# B&R Automation Studio project NAELD004C00R10L518F00 (part 51)

#### Act_LinkAction.st
```iecst
(** 2019-04-09 **)
ACTION Act_LinkAction:

	IF p_bLinkOpsRun = TRUE THEN
		//	p_eAct ACCESS p_OpsTravULMtrPshrAct;
		IF p_bLinkPullConvPullerExtCtrl
			AND p_bLinkPullConvPullerRetCtrl = FALSE
			AND p_bExtSen = FALSE
			THEN
				p_eAct := MtrPshrActExt;

		ELSIF p_bLinkPullConvPullerExtCtrl = FALSE
			AND p_bLinkPullConvPullerRetCtrl
			AND p_bRetSen = FALSE
			THEN
				p_eAct := MtrPshrActRet;

		ELSE
				p_eAct := MtrPshrActIdle;
		END_IF

	ELSIF p_bManual = TRUE THEN
//		IF p_UIMtrPshrAct = MtrPshrActStop THEN
//			p_eAct := MtrPshrActStop;
//		ELSE
			IF p_bLinkPullConvPullerExtCtrl
				AND p_bLinkPullConvPullerRetCtrl = FALSE
				AND p_bExtSen = FALSE
				THEN
				p_eAct := MtrPshrActExt;

			ELSIF p_bLinkPullConvPullerExtCtrl = FALSE
				AND p_bLinkPullConvPullerRetCtrl
				AND p_bRetSen = FALSE
				THEN
				p_eAct := MtrPshrActRet;

			ELSE
				p_eAct := MtrPshrActIdle;
			END_IF
//		END_IF

	ELSE
		p_eAct := MtrPshrActIdle;
	END_IF

END_ACTION
```

#### Act_Main.st
```iecst
(** 2019-06-17 **)
ACTION Act_Main:

	IF eStatOld <> eStat THEN
		bMtrSpdSlw	:= FALSE;

		fbMtrBrkOffDlyTm(IN := FALSE);
		fbMtrPshrExtChk(bEn := FALSE);
		fbMtrPshrRetChk(bEn := FALSE);

		IF eStatOld <> MtrPshrActIdle
			AND eStatOld <> MtrPshrActSetExt
			AND eStatOld <> MtrPshrActRstExt
			AND eStatOld <> MtrPshrActSetRet
			AND eStatOld <> MtrPshrActRstRet
			AND eStatOld <> MtrPshrActSetSpdBit0
			AND eStatOld <> MtrPshrActRstSpdBit0
			AND eStatOld <> MtrPshrActSetSpdBit1
			AND eStatOld <> MtrPshrActRstSpdBit1
			AND eStatOld <> MtrPshrActSetSpdBit2
			AND eStatOld <> MtrPshrActRstSpdBit2
			AND eStatOld <> MtrPshrActSetSigOn
			AND eStatOld <> MtrPshrActRstSigOn
			AND eStatOld <> MtrPshrActSetBrake
			AND eStatOld <> MtrPshrActRstBrake
			AND eStatOld <> MtrPshrActSetAlmRst
			AND eStatOld <> MtrPshrActRstAlmRst
			AND eStatOld <> MtrPshrActSetAll
			AND eStatOld <> MtrPshrActRstAll THEN

			bCW			:= FALSE;
			bCCW		:= FALSE;
			bSpdBinBit0	:= FALSE;
			bSpdBinBit1	:= FALSE;
			bSpdBinBit2	:= FALSE;
			bSigOn		:= FALSE;
			bBrake		:= FALSE;
			bAlmRst		:= FALSE;

		END_IF

		sStatTxt	:= a_sStatText[eStat];

		eStatOld	:= eStat;

		eStatus		:= Busy;
	END_IF

	//Main
	CASE eStat OF

		MtrPshrActIdle:
			IF EDGENEG(p_bManual) THEN
				bCW			:= FALSE;
				bCCW		:= FALSE;
				bSpdBinBit0	:= FALSE;
				bSpdBinBit1	:= FALSE;
				bSpdBinBit2	:= FALSE;
				bSigOn		:= FALSE;
				bBrake		:= FALSE;
				bAlmRst		:= FALSE;
			END_IF

			eStatus	:= Idle;

		MtrPshrActExt:
			IF eStatus = Idle OR eStatus = Busy THEN
				eStatus	:= Busy;

				//Motor Torque
				IF (p_bRetSen OR p_bRetSlowSen)AND NOT(bMtrSpdSlw) THEN
					iAnalogTorque	:= ((DINT_TO_INT(p_diStartTorque) * iMtrVolt) / 100);
				ELSIF bMtrSpdSlw THEN
					iAnalogTorque	:= ((DINT_TO_INT(p_diExtTorque) * iMtrVolt) / 100);
				END_IF

				IF iAnalogTorque < 1500 THEN
					iAnalogTorque	:= 1500;
				END_IF

				//Motor Speed
				IF p_bExtSlowSen = TRUE THEN
					bMtrSpdSlw	:= TRUE;
				END_IF

				IF bMtrSpdSlw = TRUE THEN
					diMtrSpd	:= p_diExtSlowSpd *usiPercent/100;
				ELSE
					diMtrSpd	:= p_diExtNomSpd *usiPercent/100;
				END_IF

				CASE diMtrSpd OF
					1:
						bSpdBinBit0	:= FALSE;
						bSpdBinBit1	:= FALSE;
						bSpdBinBit2	:= FALSE;
					2:
						bSpdBinBit0	:= TRUE;
						bSpdBinBit1	:= FALSE;
						bSpdBinBit2	:= FALSE;
					3:
						bSpdBinBit0	:= FALSE;
						bSpdBinBit1	:= TRUE;
						bSpdBinBit2	:= FALSE;
					4:
						bSpdBinBit0	:= TRUE;
						bSpdBinBit1	:= TRUE;
						bSpdBinBit2	:= FALSE;
					5:
						bSpdBinBit0	:= FALSE;
						bSpdBinBit1	:= FALSE;
						bSpdBinBit2	:= TRUE;
					6:
						bSpdBinBit0	:= TRUE;
						bSpdBinBit1	:= FALSE;
						bSpdBinBit2	:= TRUE;
					7:
						bSpdBinBit0	:= FALSE;
						bSpdBinBit1	:= TRUE;
						bSpdBinBit2	:= TRUE;
					8:
						bSpdBinBit0	:= TRUE;
						bSpdBinBit1	:= TRUE;
						bSpdBinBit2	:= TRUE;
				END_CASE

				//Motor On
				bSigOn	:= FALSE;
				bBrake	:= TRUE;

				IF p_bDir = TRUE THEN
					bCW		:= TRUE;
				ELSE
					bCCW	:= TRUE;
				END_IF

				//Checking Extend
				fbMtrPshrExtChk.bExtSen		:= p_bExtSen;
				fbMtrPshrExtChk.bRetSen		:= p_bRetSen;
				fbMtrPshrExtChk.bExtSafety	:= p_bExtSafetySen;

				fbMtrPshrExtChk(bEn := TRUE);

				IF fbMtrPshrExtChk.udiStatus = 0 THEN

					bSigOn	:= TRUE;
					bBrake	:= FALSE;
					bCW		:= FALSE;
					bCCW	:= FALSE;

					fbMtrBrkOffDlyTm(IN := TRUE);

					IF fbMtrBrkOffDlyTm.Q = TRUE THEN
						fbMtrBrkOffDlyTm(IN := FALSE);

						bCW			:= FALSE;
						bCCW		:= FALSE;
						bSpdBinBit0	:= FALSE;
						bSpdBinBit1	:= FALSE;
						bSpdBinBit2	:= FALSE;
						bSigOn		:= FALSE;
						bBrake		:= FALSE;

						bExtended	:= TRUE;
						eStatus		:= Done;
					END_IF

				ELSIF fbMtrPshrExtChk.udiStatus < 65534 THEN

					bCW			:= FALSE;
					bCCW		:= FALSE;
					bSpdBinBit0	:= FALSE;
					bSpdBinBit1	:= FALSE;
					bSpdBinBit2	:= FALSE;
					bSigOn		:= TRUE;
					bBrake		:= FALSE;

					bExtended	:= FALSE;
					eStatus		:= Error;

					IF fbMtrPshrExtChk.udiStatus = 1506 THEN
						udiStatus	:= 10000;	//Pusher Retract Sensor Off Time Out In Extend Check While Pusher Extend
					ELSIF fbMtrPshrExtChk.udiStatus = 1503 THEN
						udiStatus	:= 10001;	//Pusher Extend Sensor On Time Out In Extend Check While Pusher Extend
					ELSIF fbMtrPshrExtChk.udiStatus = 1507 THEN
						udiStatus	:= 10002;	//Pusher Extend Safety Sensor Error In Extend Check While Pusher Extend
					ELSE
						udiStatus	:= fbMtrPshrExtChk.udiStatus;
					END_IF

				END_IF

			END_IF

		MtrPshrActRet:
			IF eStatus = Idle OR eStatus = Busy THEN
				eStatus	:= Busy;

				//Motor Torque
				IF (p_bExtSen OR p_bExtSlowSen) AND NOT(bMtrSpdSlw) THEN
					iAnalogTorque	:= ((DINT_TO_INT(p_diStartTorque) * iMtrVolt) / 100); //32767 ==10V ,10000 == 3v
				ELSIF bMtrSpdSlw THEN
				//	iAnalogTorque	:= ((DINT_TO_INT(p_diRetTorque) * iMtrVolt) / 100);
					iAnalogTorque	:= iRetSlwTor; //6700
				END_IF

				IF iAnalogTorque < 1500 THEN
					iAnalogTorque	:= 1500;
				END_IF

				//Motor Speed
				IF p_bRetSlowSen = TRUE THEN
					bMtrSpdSlw	:= TRUE;
				END_IF

				IF bMtrSpdSlw = TRUE THEN
					diMtrSpd	:= p_diRetSlowSpd *usiPercent/100;
				ELSE
					diMtrSpd	:= p_diRetNomSpd *usiPercent/100;
				END_IF

				CASE diMtrSpd OF
					1:
						bSpdBinBit0	:= FALSE;
						bSpdBinBit1	:= FALSE;
						bSpdBinBit2	:= FALSE;
					2:
						bSpdBinBit0	:= TRUE;
						bSpdBinBit1	:= FALSE;
						bSpdBinBit2	:= FALSE;
					3:
						bSpdBinBit0	:= FALSE;
						bSpdBinBit1	:= TRUE;
						bSpdBinBit2	:= FALSE;
					4:
						bSpdBinBit0	:= TRUE;
						bSpdBinBit1	:= TRUE;
						bSpdBinBit2	:= FALSE;
					5:
						bSpdBinBit0	:= FALSE;
						bSpdBinBit1	:= FALSE;
						bSpdBinBit2	:= TRUE;
					6:
						bSpdBinBit0	:= TRUE;
						bSpdBinBit1	:= FALSE;
						bSpdBinBit2	:= TRUE;
					7:
						bSpdBinBit0	:= FALSE;
						bSpdBinBit1	:= TRUE;
						bSpdBinBit2	:= TRUE;
					8:
						bSpdBinBit0	:= TRUE;
						bSpdBinBit1	:= TRUE;
						bSpdBinBit2	:= TRUE;
				END_CASE

				//Motor On
				bSigOn	:= FALSE;
				bBrake	:= TRUE;

				IF p_bDir = TRUE THEN
					bCCW	:= TRUE;
				ELSE
					bCW		:= TRUE;
				END_IF

				//Checking Retract
				fbMtrPshrRetChk.bExtSen		:= p_bExtSen;
				fbMtrPshrRetChk.bRetSen		:= p_bRetSen;
				fbMtrPshrRetChk.bRetSafety	:= p_bRetSafetySen;

				fbMtrPshrRetChk(bEn := TRUE);

				IF fbMtrPshrRetChk.udiStatus = 0 THEN

					bSigOn	:= TRUE;
					bBrake	:= FALSE;
					bCW		:= FALSE;
					bCCW	:= FALSE;

					fbMtrBrkOffDlyTm(IN := TRUE);

					IF fbMtrBrkOffDlyTm.Q = TRUE THEN
						fbMtrBrkOffDlyTm(IN := FALSE);

						bCW			:= FALSE;
						bCCW		:= FALSE;
						bSpdBinBit0	:= FALSE;
						bSpdBinBit1	:= FALSE;
						bSpdBinBit2	:= FALSE;
						bSigOn		:= FALSE;
						bBrake		:= FALSE;

						bRetracted	:= TRUE;
						eStatus		:= Done;
					END_IF

				ELSIF fbMtrPshrRetChk.udiStatus < 65534 THEN

					bCW			:= FALSE;
					bCCW		:= FALSE;
					bSpdBinBit0	:= FALSE;
					bSpdBinBit1	:= FALSE;
					bSpdBinBit2	:= FALSE;
					bSigOn		:= TRUE;
					bBrake		:= FALSE;

					bRetracted	:= FALSE;
					eStatus		:= Error;

					IF fbMtrPshrRetChk.udiStatus = 1504 THEN
						udiStatus	:= 10003;	//Pusher Extend Sensor Off Time Out In Retract Check While Pusher Retract
					ELSIF fbMtrPshrRetChk.udiStatus = 1505 THEN
						udiStatus	:= 10004;	//Pusher Retract Sensor On Time Out In Retract Check While Pusher Retract
					ELSIF fbMtrPshrRetChk.udiStatus = 1508 THEN
						udiStatus	:= 10005;	//Pusher Retract Safety Sensor Error In Retract Check While Pusher Retract
					ELSE
						udiStatus	:= fbMtrPshrRetChk.udiStatus;
					END_IF

				END_IF

			END_IF

		MtrPshrActStop:
			IF eStatus = Idle OR eStatus = Busy THEN

				bCW			:= FALSE;
				bCCW		:= FALSE;
				bSpdBinBit0	:= FALSE;
				bSpdBinBit1	:= FALSE;
				bSpdBinBit2	:= FALSE;
				bSigOn		:= TRUE;
				bBrake		:= FALSE;

				eStatus		:= Done;

			END_IF

		MtrPshrActSetExt:
			IF eStatus = Idle OR eStatus = Busy THEN

				IF p_bDir = TRUE THEN
					bCW		:= TRUE;
				ELSE
					bCCW	:= TRUE;
				END_IF

				eStatus		:= Done;

			END_IF

		MtrPshrActRstExt:
			IF eStatus = Idle OR eStatus = Busy THEN

				IF p_bDir = TRUE THEN
					bCW		:= FALSE;
				ELSE
					bCCW	:= FALSE;
				END_IF

				eStatus		:= Done;

			END_IF

		MtrPshrActSetRet:
			IF eStatus = Idle OR eStatus = Busy THEN

				IF p_bDir = TRUE THEN
					bCCW	:= TRUE;
				ELSE
					bCW		:= TRUE;
				END_IF

				eStatus		:= Done;

			END_IF

		MtrPshrActRstRet:
			IF eStatus = Idle OR eStatus = Busy THEN

				IF p_bDir = TRUE THEN
					bCCW	:= FALSE;
				ELSE
					bCW		:= FALSE;
				END_IF

				eStatus		:= Done;

			END_IF

		MtrPshrActSetSpdBit0:
			IF eStatus = Idle OR eStatus = Busy THEN

				bSpdBinBit0	:= TRUE;

				eStatus		:= Done;

			END_IF

		MtrPshrActRstSpdBit0:
			IF eStatus = Idle OR eStatus = Busy THEN

				bSpdBinBit0	:= FALSE;

				eStatus		:= Done;

			END_IF

		MtrPshrActSetSpdBit1:
			IF eStatus = Idle OR eStatus = Busy THEN

				bSpdBinBit1	:= TRUE;

				eStatus		:= Done;

			END_IF

		MtrPshrActRstSpdBit1:
			IF eStatus = Idle OR eStatus = Busy THEN

				bSpdBinBit1	:= FALSE;

				eStatus		:= Done;

			END_IF

		MtrPshrActSetSpdBit2:
			IF eStatus = Idle OR eStatus = Busy THEN

				bSpdBinBit2	:= TRUE;

				eStatus		:= Done;

			END_IF

		MtrPshrActRstSpdBit2:
			IF eStatus = Idle OR eStatus = Busy THEN

				bSpdBinBit2	:= FALSE;

				eStatus		:= Done;

			END_IF

		MtrPshrActSetSigOn:
			IF eStatus = Idle OR eStatus = Busy THEN

				bSigOn		:= TRUE;

				eStatus		:= Done;

			END_IF

		MtrPshrActRstSigOn:
			IF eStatus = Idle OR eStatus = Busy THEN

				bSigOn		:= FALSE;

				eStatus		:= Done;

			END_IF

		MtrPshrActSetBrake:
			IF eStatus = Idle OR eStatus = Busy THEN

				bBrake		:= TRUE;

				eStatus		:= Done;

			END_IF

		MtrPshrActRstBrake:
			IF eStatus = Idle OR eStatus = Busy THEN

				bBrake		:= FALSE;

				eStatus		:= Done;

			END_IF

		MtrPshrActSetAlmRst:
			IF eStatus = Idle OR eStatus = Busy THEN

				bAlmRst		:= TRUE;

				eStatus		:= Done;

			END_IF

		MtrPshrActRstAlmRst:
			IF eStatus = Idle OR eStatus = Busy THEN

				bAlmRst		:= FALSE;

				eStatus		:= Done;

			END_IF

		MtrPshrActSetAll:
			IF eStatus = Idle OR eStatus = Busy THEN

				bCW			:= TRUE;
				bCCW		:= TRUE;
				bSpdBinBit0	:= TRUE;
				bSpdBinBit1	:= TRUE;
				bSpdBinBit2	:= TRUE;
				bSigOn		:= TRUE;
				bBrake		:= TRUE;
				bAlmRst		:= TRUE;

				eStatus		:= Done;

			END_IF

		MtrPshrActRstAll:
			IF eStatus = Idle OR eStatus = Busy THEN

				bCW			:= FALSE;
				bCCW		:= FALSE;
				bSpdBinBit0	:= FALSE;
				bSpdBinBit1	:= FALSE;
				bSpdBinBit2	:= FALSE;
				bSigOn		:= FALSE;
				bBrake		:= FALSE;
				bAlmRst		:= FALSE;

				eStatus		:= Done;

			END_IF

	END_CASE

END_ACTION
```

### WorkOrderLog.typ - Do Not Change!!!
```iecst
(*2021-06-20*)
(**)
(*Action*)
(**)

TYPE
	eWOLogAction :
		(
		WOLogActIdle,
		WOLogActDeleteOldLog,
		WOLogActCreateDir
		);
END_TYPE

(**)
```

### WorkOrderLog.var - Change By Project
```iecst
(*2019-06-10*)
(*Constant*)
(**)
(*Action & State & Status*)
VAR
	p_WOStat : UDINT;
	p_WOStatus : UDINT;
	p_WOStatTxt : UDINT;
END_VAR
(**)
(*Alarm*)
VAR
	p_WOAlmData : UDINT;
	p_WOAlmData1 : UDINT;
END_VAR
(**)
(*Output*)
```

### Program Logical/WorkOrderLog/WorkOrderLog (IEC, version 1.00.0) - 1.00.0 - NtCTSAIV v5.00.0 , NtTCP v5.00.0 , NtMessage v5.00.0

#### Init.st - Change By Project
```iecst
(** 2021-06-20 **)
PROGRAM _INIT

	(* Always Change If Project Change *)

	//Pass Address To Global Address For External Use
	//Action, State & Status
	p_WOStat	    			:= ADR(eStat);
	p_WOStatus    	   		 	:= ADR(eMainStatus);
	p_WOStatTxt      			:= ADR(sStatTxt);

	//Alarm
	p_WOAlmData      			:= ADR(tyAlmData);
	p_WOAlmData1	  			:= ADR(tyAlmData1);

	//Output

	(* Always Change If Project Change *)

END_PROGRAM
```

#### Act_InitGlobal.st - Change By Project
```iecst
(** 2021-06-20 **)
ACTION Act_InitGlobal:

	(* Always Change If Project Change *)

	p_bLinkStartupRun ACCESS p_StartupRun;

	//Pass Data To Internal Use
	p_udiRstErr ACCESS p_RstErrReset;
	//	p_bEn ACCESS p_McParamAIVEn;
	p_tyDTStructure ACCESS p_TimeCurrDTStruct;
	p_dtCurrDT ACCESS p_TimeCurrDT;

	p_bOpsRun ACCESS p_OpsRun;

	p_bNtSettingsLoadDone ACCESS p_StartupNtSettingsLoadDone;

	(* Always Change If Project Change *)
END_ACTION
```

#### InputRef_Link.var - Change By Project
```iecst
(*2021-06-20*)
(**)
(**)
VAR
	p_bLinkStartupRun : REFERENCE TO BOOL;
END_VAR
```

#### Act_LinkEn.st - Change By Project
```iecst
(** 2021-06-20 **)
ACTION Act_LinkEn:

	//Link bPrep, bEn & bDis

END_ACTION
```

#### Act_LinkAction.st - Change By Project
```iecst
(** 2021-06-20 **)
ACTION Act_LinkAction:

//	IF p_bLinkStartupRun = TRUE THEN
//		p_eAct ACCESS p_StartupCTSAct;
//	ELSE
//		p_eAct ACCESS ADR(eAct);
//	END_IF
//
END_ACTION
```

#### Act_Link.st - Change By Project
```iecst
(** 2021-06-20 **)
ACTION Act_Link:

END_ACTION
```

#### Cyclic.st - Do Not Change!!!
```iecst
(** 2021-06-20 **)
PROGRAM _CYCLIC

	IF bInitDone = FALSE THEN
		bInitDone	:= TRUE;

		Act_InitLocal;
		Act_InitGlobal;

	ELSIF bInitialDone = FALSE THEN
		IF p_bNtSettingsLoadDone = TRUE THEN
			bInitialDone	:= TRUE;

			Act_Initial;
		END_IF

	ELSE

		Act_RstErr;
		Act_LinkAction;
		Act_Action;
		Act_LinkEn;

		IF (p_bPrep = TRUE) AND (p_bEn = TRUE) AND (p_bDis = FALSE) THEN
			Act_Link;
			Act_Main;
			Act_Background;
		ELSE

			IF eStat <> WOLogActIdle THEN
				eStatus	:= Done;
			ELSE
				eStatus	:= Idle;
			END_IF
		END_IF

		Act_CombineErr;
		Act_Alarm;
		Act_Alarm1;
	END_IF

END_PROGRAM
```

#### Act_InitLocal.st - Do Not Change!!!
```iecst
(** 2021-06-20 **)
ACTION Act_InitLocal:

	//Input Reference Link To Local Variable
	p_eAct ACCESS ADR(eAct);
	p_udiRstErr ACCESS ADR(udiRstErr);
	p_bPrep ACCESS ADR(bPrep);
	p_bEn ACCESS ADR(bEn);
	p_bDis ACCESS ADR(bDis);
	p_tyDTStructure ACCESS ADR(tyDTStructure);
	p_dtCurrDT ACCESS ADR(dtCurrDT);

	p_bOpsRun ACCESS ADR(bOpsRun);

	p_udiFileKeepDay ACCESS ADR(udiFileKeepDay);
	p_sRetainFileName ACCESS ADR(sRetainFileName);
//	p_udiRetainDataAddr ACCESS ADR(udiRetainDataAddr);
//	p_udiRetainDataLen ACCESS ADR(udiRetainDataLen);
	p_sProgNm ACCESS ADR(sProgNm);

	p_bNtSettingsLoadDone ACCESS ADR(bNtSettingsLoadDone);
	p_bInternalUse ACCESS ADR(bInternalUse);

	p_sSourceString ACCESS ADR(a_sLogList);

END_ACTION
```

#### Act_RstErr.st - Do Not Change!!!
```iecst
(** 2021-06-20 **)
ACTION Act_RstErr:

	IF p_udiRstErr <> udiRstErrOld THEN
		bRstErr			:= TRUE;
		udiRstErrOld	:= p_udiRstErr;
	ELSE
		bRstErr			:= FALSE;
	END_IF

END_ACTION
```

#### Act_Action.st - Do Not Change!!!
```iecst
(** 2021-06-20 **)
ACTION Act_Action:

	//Reset Error
	IF (eStatus = Error) AND bRstErr THEN
		p_eAct	:= WOLogActIdle;
		eStat	:= WOLogActIdle;
	END_IF

	//Set p_eAct
	IF eStatus = Idle OR eStatus = Busy OR eStatus = Done THEN
		eStat	:= p_eAct;
	END_IF

END_ACTION
```

#### Act_Initial.st - Do Not Change!!!
```iecst
(** 2021-06-20 **)
ACTION Act_Initial:

	//Initial
	sStatTxt	:= a_sStatText[eStat];

	fbDirCreate1.sDevice	:= 'F';
	fbDirCreate1.sDirName	:= 'User';
	fbDirCreate1(bEn := FALSE);

	fbDirCreate2.sDevice	:= 'User';
	fbDirCreate2.sDirName	:= 'Log';
	fbDirCreate2(bEn := FALSE);

	fbDirCreate3.sDevice	:= 'Log';
	fbDirCreate3.sDirName	:= 'WorkOrderLog';
	fbDirCreate3(bEn := FALSE);

	fbFileAppend1.sDevice	        := 'CTSLog';
	fbFileAppend1(bEn := FALSE);

	fbFileAppend2.sDevice	        := 'CTSLog';
	fbFileAppend2(bEn := FALSE);

	fbFileOldDel1.sDevice			:= 'CTSLog';
	fbFileOldDel1.sPath				:= '';
	fbFileOldDel1.sKeyword			:= p_sProgNm;
	fbFileOldDel1.udiFileKeepDay	:= p_udiFileKeepDay;
	fbFileOldDel1(bEn := FALSE);

END_ACTION
```

#### Act_Main.st - Do Not Change!!!
```iecst
(** 2021-06-20 **)
ACTION Act_Main:

	IF eStatOld <> eStat THEN
		fbFileOldDel1(bEn := FALSE);
		fbDirCreate1(bEn := FALSE);
		fbDirCreate2(bEn := FALSE);
		fbDirCreate3(bEn := FALSE);
		bFileNotFound	:= FALSE;
		sStatTxt	:= a_sStatText[eStat];

		eStatOld	:= eStat;

		eStatus		:= Busy;
	END_IF

	//Main
	CASE eStat OF

		WOLogActIdle:
			eStatus	:= Idle;

		WOLogActCreateDir:
			IF eStatus = Idle OR eStatus = Busy THEN

				eStatus	:= Busy;

				sStatTxt	:= a_sStatText[eStat];

				CASE usiStep OF
					0:
						fbDirCreate1(bEn := TRUE);
						IF fbDirCreate1.udiStatus = 0 THEN
							usiStep	:= 1;
						ELSIF fbDirCreate1.udiStatus < 65534 THEN
							eStatus		:= Error;

							IF fbDirCreate1.udiStatus = 1908 THEN
								udiStatus	:= 10016;	//Create User Directory Error
							ELSE
								udiStatus	:= fbDirCreate1.udiStatus;
							END_IF
						END_IF

					1:
						fbDirCreate2(bEn := TRUE);
						IF fbDirCreate2.udiStatus = 0 THEN
							eStatus	:= Done;
						ELSIF fbDirCreate2.udiStatus < 65534 THEN
							eStatus		:= Error;

							IF fbDirCreate2.udiStatus = 1908 THEN
								udiStatus	:= 10017;	//Create CTSLog Directory Error
							ELSE
								udiStatus	:= fbDirCreate2.udiStatus;
							END_IF
						END_IF

				END_CASE

			END_IF

		WOLogActDeleteOldLog:
			IF eStatus = Idle OR eStatus = Busy THEN

				eStatus	:= Busy;

				fbFileOldDel1.dtDTNow	:= p_dtCurrDT;
				fbFileOldDel1(bEn := TRUE);
				IF fbFileOldDel1.udiStatus = 0 THEN
					eStatus	:= Done;
				ELSIF fbFileOldDel1.udiStatus < 65534 THEN
					eStatus		:= Error;

					IF fbFileOldDel1.udiStatus = 1910 THEN
						udiStatus	:= 10018;	//Get Directory Info Error While Deleting Old Log
					ELSIF fbFileOldDel1.udiStatus = 1911 THEN
						udiStatus	:= 10019;	//Directory Read Error While Deleting Old Log
					ELSIF fbFileOldDel1.udiStatus = 1912 THEN
						udiStatus	:= 10020;	//File Delete Error While Deleting Old Log
					ELSE
						udiStatus	:= fbFileOldDel1.udiStatus;
					END_IF
				END_IF

			END_IF

		ELSE
			IF eStatus = Idle OR eStatus = Busy THEN
				eStatus	:= Done;
			END_IF

	END_CASE

END_ACTION
```

#### Act_Background.st - Do Not Change!!!
```iecst
(** 2021-06-20 **)
ACTION Act_Background:

	Act_Background_Log;

	//Reset Error

	IF (eStatus1 = Error) AND bRstErr THEN
		eStatus1	:= Idle;
		udiStatus1	:= 0;

		fbFileAppend1(bEn := FALSE);
		i	:= 0;

	END_IF

END_ACTION
```

#### Act_Background_Log.st - Do Not Change!!!
```iecst
(** 2021-06-20 **)
ACTION Act_Background_Log:
	if
	IF eStatus1 <> Error THEN
		IF udiWriteLogCntr <> udiLogCntr THEN

			CASE i OF

				0:
					dtCurrDTTemp			:= p_dtCurrDT;
					fbFileAppend1.sFile		:= DT_TO_STRING(dtCurrDTTemp);
					fbFileAppend1.sFile		:= MID(fbFileAppend1.sFile , 10 , 4);
					fbFileAppend1.sFile		:= CONCAT(p_sProgNm , fbFileAppend1.sFile);
					fbFileAppend1.sFile		:= CONCAT(fbFileAppend1.sFile , '.dat');

					fbFileAppend1.p_Src		:= ADR(p_sSourceString);
					fbFileAppend1.udiLen	:= LEN(p_sSourceString);

					i	:= 1;

				1:
					fbFileAppend1(bEn := TRUE);
					IF fbFileAppend1.udiStatus = 0 THEN
						fbFileAppend1(bEn := FALSE);

						udiWriteLogCntr	:= udiWriteLogCntr + 1;
						IF udiWriteLogCntr = 10 THEN
							udiWriteLogCntr	:= 0;
						END_IF

						i	:= 0;

					ELSIF fbFileAppend1.udiStatus < 65534 THEN
						eStatus1	:= Error;

						IF fbFileAppend1.udiStatus = 1900 THEN
							udiStatus1	:= 10000;	//File Open Error While Writing Log
						ELSIF fbFileAppend1.udiStatus = 1901 THEN
							udiStatus1	:= 10001;	//File Create Error While Writing Log
						ELSIF fbFileAppend1.udiStatus = 1913 THEN
							udiStatus1	:= 10002;	//Get File Info Error While Writing Log
						ELSIF fbFileAppend1.udiStatus = 1903 THEN
							udiStatus1	:= 10003;	//File Write Error While Writing Log
						ELSIF fbFileAppend1.udiStatus = 1904 THEN
							udiStatus1	:= 10004;	//File Close Error While Writing Log
						ELSIF fbFileAppend1.udiStatus = 1914 THEN
							udiStatus1	:= 10005;	//Directory Does Not Exist While Writing Log
						ELSE
							udiStatus1	:= fbFileAppend1.udiStatus;
						END_IF

						i	:= 0;
					END_IF
			END_CASE
		END_IF

END_ACTION
```

#### Act_CombineErr.st - Do Not Change!!!
```iecst
(** 2021-06-20 **)
ACTION Act_CombineErr:

	//Combine Error
	IF eStatus = Error OR eStatus1 = Error THEN
		eMainStatus	:= Error;
	ELSE
		eMainStatus	:= eStatus;
	END_IF

END_ACTION
```

#### Act_Alarm.st - Do Not Change!!!
```iecst
(** 2021-06-20 **)
ACTION Act_Alarm: //eStatus for Act_Main.st

	//Error
	IF EDGEPOS(eStatus = Error) THEN

		tyAlmData.sProgNm		:= p_sProgNm;
		tyAlmData.udiCode		:= udiStatus;
		tyAlmData.eSeverity		:= AlmSeverityError;
		tyAlmData.udiRunTime	:= tyAlmData.udiRunTime + 1;

		//Get Error Message
		IF tyAlmData.udiCode < 10000 OR tyAlmData.udiCode > 10199 THEN
			tyAlmData.sAlmMsg	:= 'Unknown';
			tyAlmData.sRcyMsg	:= 'Unknown';
		ELSE
			tyAlmData.sAlmMsg	:= a_tyAlmText[tyAlmData.udiCode].sAlmText;
			tyAlmData.sRcyMsg	:= a_tyAlmText[tyAlmData.udiCode].sRcyText;
		END_IF

		sStatTxt	:= tyAlmData.sAlmMsg;

	ELSIF bRstErr AND (tyAlmData.udiCode <> 0) THEN

		tyAlmData.udiCode	:= 0;
		tyAlmData.eSeverity	:= AlmSeverityNA;
		tyAlmData.sAlmMsg	:= '';
		tyAlmData.sRcyMsg	:= '';

		sStatTxt	:= a_sStatText[eStat];

	END_IF

END_ACTION
```

#### Act_Alarm1.st - Do Not Change!!!
```iecst
(** 2021-06-20 **)
ACTION Act_Alarm1: //eStatus1 for General Error like Sequence Error, CreateSvr Error, TCP Error and etc.

	//Error
	IF EDGEPOS(eStatus1 = Error) THEN

		tyAlmData1.sProgNm		:= p_sProgNm;
		tyAlmData1.udiCode		:= udiStatus1;
		tyAlmData1.eSeverity	:= AlmSeverityError;
		tyAlmData1.udiRunTime	:= tyAlmData1.udiRunTime + 1;

		//Get Error Message
		IF tyAlmData1.udiCode < 10000 OR tyAlmData1.udiCode > 10199 THEN
			tyAlmData1.sAlmMsg	:= 'Unknown';
			tyAlmData1.sRcyMsg	:= 'Unknown';
		ELSE
			tyAlmData1.sAlmMsg	:= a_tyAlmText[tyAlmData1.udiCode].sAlmText;
			tyAlmData1.sRcyMsg	:= a_tyAlmText[tyAlmData1.udiCode].sRcyText;
		END_IF

		sStatTxt	:= tyAlmData1.sAlmMsg;

	ELSIF bRstErr AND (tyAlmData1.udiCode <> 0) THEN

		tyAlmData1.udiCode		:= 0;
		tyAlmData1.eSeverity	:= AlmSeverityNA;
		tyAlmData1.sAlmMsg		:= '';
		tyAlmData1.sRcyMsg		:= '';

		sStatTxt	:= a_sStatText[eStat];

	END_IF

END_ACTION
```

#### InputRef.var - Do Not Change!!!
```iecst
(*2019-06-10*)
(**)
(*General*)
VAR
	p_eAct : REFERENCE TO eWOLogAction;
	p_udiRstErr : REFERENCE TO UDINT;
	p_bPrep : REFERENCE TO BOOL;
	p_bEn : REFERENCE TO BOOL;
	p_bDis : REFERENCE TO BOOL;
END_VAR
(**)
(*Configuration*)
VAR
	p_tyDTStructure : REFERENCE TO DTStructure;
	p_dtCurrDT : REFERENCE TO DATE_AND_TIME;
END_VAR
(**)
(*Input*)
VAR
	p_udiSndBffrSize : REFERENCE TO UDINT;
	p_udiRcvBffrSize : REFERENCE TO UDINT;
	p_bOpsRun : REFERENCE TO BOOL;
	p_udiFileKeepDay : REFERENCE TO UDINT;
	p_udiRetainDataAddr : REFERENCE TO UDINT;
	p_udiRetainDataLen : REFERENCE TO UDINT;
	p_sRetainFileName : REFERENCE TO STRING[80];
	p_usiAliveReqCntr : REFERENCE TO USINT;
	p_udiAliveIdleTimeInSec : REFERENCE TO UDINT;
	p_tAliveRcvTimeOut : REFERENCE TO TIME;
	p_tSendLaneInfoResTm : REFERENCE TO TIME;
	p_diTransferInTO : REFERENCE TO DINT;
	p_sProgNm : REFERENCE TO STRING[15];
	p_sSourceString : REFERENCE TO STRING[80];
	p_bNtSettingsLoadDone : REFERENCE TO BOOL;
END_VAR
```

#### Local.var - Do Not Change!!!
```iecst
(*2019-06-10*)
(**)
(*Local Action, State & Status*)
VAR
	eAct : eWOLogAction := WOLogActIdle;
	eStat : eWOLogAction := WOLogActIdle;
	eMainStatus : eFBStatus := Idle;
	eStatus : eFBStatus := Idle;
	eStatus1 : eFBStatus := Idle;
	udiStatus : UDINT := 0;
	udiStatus1 : UDINT := 0;
	sStatTxt : STRING[200] := '';
	a_sStatText : ARRAY[0..50] OF STRING[200] := ['Idling','Background Starting Operations','Background Stopping Operations','Deleting Old Log File','Creating Directory','Writing Retain File','Reading Retain File','Saving Configuration',43('')];
END_VAR
(**)
(*Local Alarm*)
VAR
	tyAlmData : tyAlmDat;
	tyAlmData1 : tyAlmDat;
	a_tyAlmText : {REDUND_UNREPLICABLE} ARRAY[10000..10199] OF tyAlmTxt := [(sAlmText:='File Open Error While Writing Log',sRcyText:='An Error Was Encountered While Trying To Open File. Please Contact Nutek For A Possible Solution.'),(sAlmText:='File Create Error While Writing Log',sRcyText:='An Error Was Encountered While Trying To Create File. Please Contact Nutek For A Possible Solution.'),(sAlmText:='Get File Info Error While Writing Log',sRcyText:='An Error Was Encountered While Getting File Info. Please Contact Nutek For A Possible Solution.'),(sAlmText:='File Write Error While Writing Log',sRcyText:='An Error Was Encountered While Trying To Write File. Please Contact Nutek For A Possible Solution.'),(sAlmText:='File Close Error While Writing Log',sRcyText:='An Error Was Encountered While Trying To Close File. Please Contact Nutek For A Possible Solution.'),(sAlmText:='Directory Does Not Exist While Writing Log',sRcyText:='The Directory Does Not Exist.Please Contact Nutek For A Possible Solution.'),(sAlmText:='Invalid Ident While Closing TCP',sRcyText:='Invalid Ident Value.'),(sAlmText:='Closing TCP Error',sRcyText:='Problem Occurred In The TCP/IP Connection. Check The Connection And Try To Reconnect.'),0,(sAlmText:='Board Jam At Sensor After Transfer Interrupted',sRcyText:='Pull Back Board From Downstream Machine'),0,(sAlmText:='Send Board Info Request To Send From Upstream Hermes',sRcyText:='Sending Illegal Message.'),(sAlmText:='Query Work Order Info Request To Send From Upstream Hermes',sRcyText:='Sending Illegal Message.'),(sAlmText:='Send Work Order Info Request To Send From Upstream Hermes',sRcyText:='Sending Illegal Message.'),(sAlmText:='Board Arrived Request To Send From Upstream Hermes',sRcyText:='Sending Illegal Message.'),(sAlmText:='Board departed Request To Send From Upstream Hermes',sRcyText:='Sending Illegal Message.'),(sAlmText:='Forecast Id Mismatch While Checking BoardForecast & Machine Ready',sRcyText:='The ForecastId Value Does Not Match. Change The Value And Resend The Value.'),(sAlmText:='Product Type Id Mismatch While Checking BoardForecast & Machine Ready',sRcyText:='The ProductTypetId Value Does Not Match. Change The Value And Resend The Value.'),(sAlmText:='Width Mismatch While Checking BoardForecast & Machine Ready',sRcyText:='The Width Value Does Not Match. Change The Value And Resend The Value.'),(sAlmText:='Query Top Barcode and Bottom Barcode found from different Recipes',sRcyText:='Please Check or Scan Again the PCB Barcode'),32(0)];
END_VAR
(**)
(*Local Output*)
VAR
	bConnected : BOOL;
	bHandshakeDone : BOOL;
END_VAR
(**)
(*Local Input*)
VAR
	udiRstErr : UDINT := 0;
	bPrep : BOOL := TRUE;
	bEn : BOOL := TRUE;
	bDis : BOOL := FALSE;
	usiStep : USINT;
	uiSvrPort : UINT := 51111;
	uiSvrPortOld : UINT;
	sIPAddr : STRING[15] := '192.168.0.100';
	tyDTStructure : DTStructure := (year:=2020,month:=11,day:=11,wday:=05,hour:=21,minute:=28,second:=30,millisec:=123,microsec:=456);
	dtCurrDT : DATE_AND_TIME := DT#2019-02-23-12:30:50;
	udiSndBffrSize : UDINT := 65536;
	udiRcvBffrSize : UDINT := 65536;
	udiAliveIdleTimeInSec : UDINT := 5;
	tAliveRcvTimeOut : TIME := T#5S;
	bOpsRun : BOOL := FALSE;
	udiFileKeepDay : UDINT := 30;
	sRetainFileName : STRING[80] := 'WorkOrderLog.dat';
	sProgNm : STRING[15] := 'WorkOrderLog';
	bNtSettingsLoadDone : BOOL := TRUE;
END_VAR
(**)
(*Local*)
VAR
	sMsg : STRING[80];
	bRstErr : BOOL;
	udiRstErrOld : UDINT;
	bInitDone : BOOL;
	bInitialDone : BOOL;
	bRun : BOOL;
	bStop : BOOL;
	bRstConnection : BOOL;
	bRstState : BOOL;
	fbCreateSvr : fbTCPCreateSvr;
	fbDirCreate1 : fbDirCreate;
	fbDirCreate2 : fbDirCreate;
	fbDirCreate3 : fbDirCreate;
	i : UDINT := 0;
	j : UDINT := 0;
	jj : UDINT := 0;
	udiLogCntrSnd : UDINT := 1;
	udiWriteLogCntrSnd : UDINT := 1;
	a_sLogListSnd : ARRAY[1..10] OF STRING[65535];
	udiLogCntrRcv : UDINT := 1;
	udiWriteLogCntrRcv : UDINT := 1;
	a_sLogListRcv : ARRAY[1..10] OF STRING[65535];
	sDT : STRING[80];
	dtCurrDTTemp : DATE_AND_TIME;
	fbFileAppend1 : fbFileFullAppend;
	fbFileOldDel1 : fbFileOldDel;
	fbFileRead1 : fbFileFullRead;
	fbFileWrite1 : fbFileFullWrite;
	bFileNotFound : BOOL;
	udiWriteLogCntr : UDINT;
	udiLogCntr : UDINT;
	a_sLogList : ARRAY[0..c_udiFrmHistoryMax] OF STRING[200];
END_VAR
(**)
(**)
```

### AutoRcp.var - Change By Project
```iecst
(*2019-06-27*)
(**)
(*Action & State & Status*)
VAR
	p_AutoRcpStat : UDINT;
	p_AutoRcpStatus : UDINT;
END_VAR
(**)
(*Alarm*)
VAR
	p_AutoRcpAlmData : UDINT;
	p_AutoRcpInfoData : UDINT;
	p_AutoRcpInfoData1 : UDINT;
END_VAR
(**)
(*Output*)
VAR
	p_AutoRcpUSAllow : UDINT;
	p_AutoRcpDSAllow : UDINT;
	p_AutoRcpProdAccDataMnl : UDINT;
	p_AutoRcpProdUpdtDataMnl : UDINT;
	p_AutoRcpMagAccDataMnl : UDINT;
	p_AutoRcpTimeAct : UDINT;
	p_AutoRcpSetDT : UDINT;
	p_AutoRcpWaitRlsBrd : UDINT;
	p_AutoRcpUpdtProdRcp : UDINT;
	p_AutoRcpProdRcpDiff : UDINT;
	p_AutoRcpCurrRcpProdID : UDINT;
	p_AutoRcpCurrRcpWidth : UDINT;
	p_AutoRcpCurrDeleteSendWO : UDINT;
	p_AutoRcpbTravWidthDiffblk : UDINT;
	p_AutoRcpbMagChangeOverBlk : UDINT;
	p_AutoRcpbMag1PropDiffBlk : UDINT;
	p_AutoRcpbMag2PropDiffBlk : UDINT;
	p_AutoRcpbMag3PropDiffBlk : UDINT;
	p_AutoRcpbMag1WidthChg : UDINT;
	p_AutoRcpbMag2WidthChg : UDINT;
	p_AutoRcpbMag3WidthChg : UDINT;
END_VAR
(*TravLif Width*)
VAR
	p_AutoRcpTravLifWidth : UDINT;
	p_AutoRcpTravLifPitch : UDINT;
END_VAR
(*MagConv*)
VAR
	p_AutoRcpbMag1RcpLoaded : UDINT;
	p_AutoRcpbMag2RcpLoaded : UDINT;
	p_AutoRcpbMag3RcpLoaded : UDINT;
	p_AutoRcpTravLif : UDINT;
	p_AutoRcpMagRcp : UDINT;
	p_AutoRcpWorkOrderId : UDINT;
	p_AutoRcpFollower1 : UDINT;
END_VAR
(*Magazine Properties*)
VAR
	p_diAutoRcpMag1MaxSlt : UDINT;
	p_diAutoRcpMag1MinSlt : UDINT;
	p_diAutoRcpMag1Pitch : UDINT;
	p_diAutoRcpMag1Width : UDINT;
	p_diAutoRcpMag2MaxSlt : UDINT;
	p_diAutoRcpMag2MinSlt : UDINT;
	p_diAutoRcpMag2Pitch : UDINT;
	p_diAutoRcpMag2Width : UDINT;
	p_diAutoRcpMag3MaxSlt : UDINT;
	p_diAutoRcpMag3MinSlt : UDINT;
	p_diAutoRcpMag3Pitch : UDINT;
	p_diAutoRcpMag3Width : UDINT;
END_VAR
```

### Program Logical/AutoRcp/AutoRcp (IEC, version 1.00.0) - 1.00.0 - NtHermes v5.00.0 , NtTCP v5.00.0 , NtMessage v5.00.0

#### Init.st - Change By Project
```iecst
(** 2019-06-27 **)
PROGRAM _INIT

	(* Always Change If Project Change *)

	//Physical Configuration
	bAutoUpdtData	:= TRUE;
	bInternalUse	:= TRUE;

	//Pass Address To Global Address For External Use
	//Action, State & Status
	p_AutoRcpStat		:= ADR(eStat);
	p_AutoRcpStatus	:= ADR(eStatus);

	//Alarm
	p_AutoRcpAlmData		:= ADR(tyAlmData);
	p_AutoRcpInfoData		:= ADR(tyInfoData);
	p_AutoRcpInfoData1	:= ADR(tyInfoData1);

	//Output
//	p_AutoRcpUSAllow			:= ADR(bUSAllow);
//	p_AutoRcpDSAllow			:= ADR(bDSAllow);

	p_AutoRcpCurrRcpProdID	:= ADR(sProdtypeID);
	p_AutoRcpCurrRcpWidth :=  ADR(diProdWidth);
	p_AutoRcpCurrDeleteSendWO :=  ADR(bDeleteSendWO); //svyhermes

	p_AutoRcpbTravWidthDiffblk := ADR(bTravLifWidthDiffBlk);

	(*p_AutoRcp:= ADR(a_bCheckDifferent);*)
	p_AutoRcpbMag1PropDiffBlk := ADR(a_bCheckDifferent[1]);
	p_AutoRcpbMag2PropDiffBlk := ADR(a_bCheckDifferent[2]);
	p_AutoRcpbMag3PropDiffBlk := ADR(a_bCheckDifferent[3]);

	p_AutoRcpbMagChangeOverBlk := ADR(a_bMagChangOverBlk);

	p_AutoRcpbMag1WidthChg	:= ADR (a_bAllwChangeWidth[1]);
	p_AutoRcpbMag2WidthChg	:= ADR (a_bAllwChangeWidth[2]);
	p_AutoRcpbMag3WidthChg	:= ADR (a_bAllwChangeWidth[3]);

	p_AutoRcpbMag1RcpLoaded	:= ADR (a_bRcpLoaded[1]); //to opsMagConv
	p_AutoRcpbMag2RcpLoaded	:= ADR (a_bRcpLoaded[2]);
	p_AutoRcpbMag3RcpLoaded	:= ADR (a_bRcpLoaded[3]);

	p_AutoRcpTravLifWidth := ADR(diTravLifWidth);
	p_AutoRcpTravLifPitch := ADR(diTravLifPitch);

	p_diAutoRcpMag1MaxSlt  := ADR(a_tyMagProps[1].diMaxSlt); //to buffer ,UI display
	p_diAutoRcpMag1MinSlt  := ADR(a_tyMagProps[1].diMinSlt);
	p_diAutoRcpMag1Pitch   := ADR(a_tyMagProps[1].diPitch);
	p_diAutoRcpMag1Width   := ADR(a_tyMagProps[1].diWidth);

	p_diAutoRcpMag2MaxSlt  := ADR(a_tyMagProps[2].diMaxSlt);
	p_diAutoRcpMag2MinSlt  := ADR(a_tyMagProps[2].diMinSlt);
	p_diAutoRcpMag2Pitch   := ADR(a_tyMagProps[2].diPitch);
	p_diAutoRcpMag2Width   := ADR(a_tyMagProps[2].diWidth);

	p_diAutoRcpMag3MaxSlt  := ADR(a_tyMagProps[3].diMaxSlt);
	p_diAutoRcpMag3MinSlt  := ADR(a_tyMagProps[3].diMinSlt);
	p_diAutoRcpMag3Pitch   := ADR(a_tyMagProps[3].diPitch);
	p_diAutoRcpMag3Width   := ADR(a_tyMagProps[3].diWidth);

	p_AutoRcpTravLif	 	:= ADR(tyCurrZ1Rcp);
	p_AutoRcpMagRcp		 	:= ADR(a_tyCurrZ2Rcp);
	p_AutoRcpWorkOrderId	 := ADR(sWorkOrderId);
	p_AutoRcpFollower1		 := ADR(a_tyAutoRcpFollower1);
	(* Always Change If Project Change *)

END_PROGRAM
```

#### Package Logical/AutoRcp/AutoRcp/PrecededBySelf_Hermes - Intended for F1,F2

#### PrecededBySelfBackground1.st
```iecst
ACTION PrecededBySelfBackground1:

//Converting BA from US Hermes to Rcp
	IF EDGEPOS(p_bSndWorkOrderInfo) THEN
		tyCurrReqRcp.sBoardId := p_tySendWorkOrderData.tyData.sBoardId;
		tyCurrReqRcp.sBoardIdCreatedBy := p_tySendWorkOrderData.tyData.sBoardIdCreatedBy;
		tyCurrReqRcp.eFailedBoard := p_tySendWorkOrderData.tyData.eFailedBoard;
		tyCurrReqRcp.sProductTypeId := p_tySendWorkOrderData.tyData.sProductTypeId;
		tyCurrReqRcp.eFlippedBoard := p_tySendWorkOrderData.tyData.eFlippedBoard;
		tyCurrReqRcp.sTopBarcode := p_tySendWorkOrderData.tyData.sTopBarcode;
		tyCurrReqRcp.sBottomBarcode := p_tySendWorkOrderData.tyData.sBottomBarcode;
		tyCurrReqRcp.rLength := p_tySendWorkOrderData.tyData.rLength;
		tyCurrReqRcp.rWidth := p_tySendWorkOrderData.tyData.rWidth;
		tyCurrReqRcp.rThickness := p_tySendWorkOrderData.tyData.rThickness;
		tyCurrReqRcp.rConveyorSpeed := p_tySendWorkOrderData.tyData.rConveyorSpeed;
		tyCurrReqRcp.rTopClearanceHeight := p_tySendWorkOrderData.tyData.rTopClearanceHeight;
		tyCurrReqRcp.rBottomClearanceHeight := p_tySendWorkOrderData.tyData.rBottomClearanceHeight;
		tyCurrReqRcp.rWeight := p_tySendWorkOrderData.tyData.rWeight;
		tyCurrReqRcp.sWorkOrderId := p_tySendWorkOrderData.tyData.sWorkOrderId;
		tyCurrReqRcp.sBatchId := p_tySendWorkOrderData.tyData.sBatchId;

	END_IF

	//Error Handling
	IF p_bLinkOpsRun AND p_bSndWorkOrderInfo THEN
		IF tyCurrReqRcp.rWidth < DINT_TO_REAL(p_diNtParamProdRcpMinWidth)/1000.0 THEN
			eStatus := Error;
			udiStatus := 10010;
		ELSIF tyCurrReqRcp.rWidth  > DINT_TO_REAL(p_diNtParamProdRcpMaxWidth)/1000.0 THEN
			eStatus := Error;
			udiStatus := 10011;
		ELSIF  tyCurrReqRcp.rThickness  > DINT_TO_REAL(p_tyNtParamAutoRcpParamLmt.diThicknessInUM)/1000.0 THEN
			eStatus := Error;
			udiStatus := 10012;
		ELSIF  tyCurrReqRcp.rBottomClearanceHeight  > DINT_TO_REAL(p_tyNtParamAutoRcpParamLmt.diMaxBottomCleranceInUM)/1000.0 THEN
			eStatus := Error;
			udiStatus := 10013;
		ELSIF tyCurrReqRcp.rTopClearanceHeight > DINT_TO_REAL(p_tyNtParamAutoRcpParamLmt.diMaxTopClearamceInUM)/1000.0 THEN
			eStatus := Error;
			udiStatus := 10014;
		END_IF
		IF tyCurrReqRcp.rBottomClearanceHeight <= 5.5 AND p_diNtParamPullerHeightInMM <= 19 THEN
			p_diRequestedMinSlt := 3;
		ELSE
			p_diRequestedMinSlt := 6;
		END_IF

		IF eStatus = Error THEN
			p_ausiSvyMagAccOrder[p_usiSvyMagOrderPos] := 0;  //bi-dir
			p_asSvyHermesMagGUID[p_usiSvyMagOrderPos] := ''; //bi-dir
			IF p_usiSvyMagOrderPos = 1 THEN
				p_bLinkOpsMagConvLD1QueryWO := FALSE; //bi-dir ,cancel bQueryWO
			ELSIF p_usiSvyMagOrderPos =2 THEN
				p_bLinkOpsMagConvLD2QueryWO := FALSE; //bi-dir
			ELSIF p_usiSvyMagOrderPos =3 THEN
				p_bLinkOpsMagConvLD3QueryWO := FALSE; //bi-dir
			END_IF
			p_usiSvyMagOrderPos := 0;	  //bi-dir
			p_bSndWorkOrderInfo := FALSE; //bi-dir
		END_IF

		//Delete sendWorkOrder
		bDeleteSendWO := TRUE;
	END_IF

	//For Zone 1 Initialization Only (follow internal rcp width)
	IF bInitializedFollower1Done = FALSE THEN
		IF p_tyInternalReqProdRcp.diWidthInUM <> 0 THEN
			tyCurrZ1Rcp.rWidth := p_tyInternalReqProdRcp.diWidthInUM/1000 ; //Z1Rcp == TravLif
			bOverWriteTravLifProperties := TRUE;
			bInitializedFollower1Done := TRUE;
		END_IF
	END_IF

	IF p_usiSvyMagOrderPos > 0 AND eStatus <> Error THEN
		a_tyCurrZ2Rcp[p_usiSvyMagOrderPos] := tyCurrReqRcp;
		bOverWriteMagProperties := TRUE;
		usiChg := usiChg + 1;
		p_usiSvyMagOrderPos := 0;	  //bi-dir
		p_bSndWorkOrderInfo := FALSE; //bi-dir
	END_IF

	//Follower1 //Changed to a_tyCurrZ2Rcp //Assign when received WO and empty rcp
	FOR usi := 1 TO 3 DO
		IF p_ausiSvyMagAccOrder[usi] = 10 AND eStatus <> Error THEN
			IF memcmp(ADR(a_tyCurrZ2Rcp[usi]) , ADR(tyCurrZ1Rcp) , SIZEOF(a_tyCurrZ2Rcp[usi])) <> 0 THEN
				bTravLifWidthDiffBlk := TRUE; //block travlif USallow
				IF p_bZ1AccNewRcpCondition THEN
					tyCurrZ1Rcp := a_tyCurrZ2Rcp[usi];
					//a_tyCurrZ2Rcp[usi] := tyCurrReqRcp;
					//bOverWriteTravLifProperties := TRUE;
					//bOverWriteMagProperties := TRUE;
					//usiChg := usiChg + 1;
					//p_bSndWorkOrderInfo := FALSE; //bi-dir
				END_IF
			ELSE
				bTravLifWidthDiffBlk := FALSE;
			END_IF
		END_IF
	END_FOR

	//IF all was block with magazine available then Force the Magazine Exit
	FOR ii:= 1 TO SIZEOF(a_bMagChangOverBlk)/SIZEOF(a_bMagChangOverBlk[1]) DO
		IF  (a_bBufferMagPresent[ii] AND a_bMagChangOverBlk[ii] = FALSE) OR NOT(a_bBufferMagPresent[ii]) THEN
			EXIT;
		END_IF
	END_FOR
	IF ii = SIZEOF(a_bMagChangOverBlk)/SIZEOF(a_bMagChangOverBlk[1]) THEN
		bForceExitMag := TRUE; //force Magazine to exit the highest priority Mag
	ELSE
		bForceExitMag := FALSE;
	END_IF

END_ACTION
```

#### PrecededBySelfBackground2.st
```iecst
ACTION PrecededBySelfBackground2:

	//Convert ProdID to Rcp Name and rWidth to diWidth for F0 to output Hermes
//	sProdtypeID:= tyCurrReqRcp.sProductTypeId;
//	diProdWidth := REAL_TO_DINT(tyCurrReqRcp.rWidth*1000);

	//Convert to Width for F1 //Changed to a_tyCurrZ2Rcp
//	IF bOverWriteTravLifProperties THEN
	IF p_ausiSvyMagAccOrder[1] = 0 AND p_ausiSvyMagAccOrder[2] = 0 AND p_ausiSvyMagAccOrder[3] = 0 THEN
		diTravLifWidth := 100000;
	ELSE
		FOR usi := 1 TO 3 DO
			IF p_ausiSvyMagAccOrder[usi] = 10 AND p_bConvHvBrd = FALSE THEN
				tyCurrZ1Rcp := a_tyCurrZ2Rcp[usi];
				rPitch := (tyCurrZ1Rcp.rTopClearanceHeight + tyCurrZ1Rcp.rBottomClearanceHeight + tyCurrZ1Rcp.rThickness)/(p_diMagRcpCurrRcpSltToSlt/1000);
				diTravLifPitch := REAL_TO_DINT(ceil(rPitch));
				diTravLifWidth := REAL_TO_DINT(tyCurrZ1Rcp.rWidth*1000);
				sWorkOrderId	:= tyCurrZ1Rcp.sWorkOrderId;	//to DSHermes
				EXIT;
				//diTravLifWidth := REAL_TO_DINT(a_tyCurrZ2Rcp[usi].rWidth*1000);
			END_IF
		END_FOR
	END_IF
	//		bOverWriteTravLifProperties	:= FALSE;
	//	END_IF

	//Convert to Pitch for F2
	IF bOverWriteMagProperties = TRUE THEN
		IF p_bProdSelTopToBtm THEN
			//overwriting diMax
			FOR kk := 1 TO 3 DO//SIZEOF(a_tyCurrZ2Rcp)/SIZEOF(a_tyCurrZ2Rcp[1]) DO //top to btm
				rMinslt :=  (a_tyCurrZ2Rcp[kk].rBottomClearanceHeight)/(p_diMagRcpCurrRcpSltToSlt/1000);
				rMaxslt := (p_diMagRcpCurrRcpTtlSlt-p_diRequestedMinSlt) - ((a_tyCurrZ2Rcp[kk].rTopClearanceHeight + a_tyCurrZ2Rcp[kk].rThickness)/(p_diMagRcpCurrRcpSltToSlt/1000)) + 1;
				rPitch := (a_tyCurrZ2Rcp[kk].rTopClearanceHeight + a_tyCurrZ2Rcp[kk].rBottomClearanceHeight + a_tyCurrZ2Rcp[kk].rThickness)/(p_diMagRcpCurrRcpSltToSlt/1000);

				rNumInterval := (rMaxslt - rMinslt )/ceil(rPitch);
				diCalcedMax := REAL_TO_DINT(floor(rMaxslt));
				diCalcedPitch := REAL_TO_DINT(ceil(rPitch));
				diCalcedMin := REAL_TO_DINT((diCalcedMax - floor(rNumInterval)*ceil(rPitch)));

				IF diCalcedMin = 0 THEN
					diCalcedMin := diCalcedPitch;
				END_IF
				//			IF diCalcedMin < p_diRequestedMinSlt THEN
				//				diModulus :=  p_diRequestedMinSlt/diCalcedMin;
				//				diCalcedMin := diCalcedMin + diModulus*diCalcedPitch;
				//			END_IF
				a_tyMagProps[kk].diMaxSlt := diCalcedMax;
				a_tyMagProps[kk].diMinSlt := diCalcedMin;
				a_tyMagProps[kk].diPitch  := diCalcedPitch;
				a_tyMagProps[kk].diWidth := REAL_TO_DINT(a_tyCurrZ2Rcp[kk].rWidth * 1000);
				IF a_tyCurrZ2Rcp[kk].sWorkOrderId <> '' AND diCalcedMin <> 0 AND p_ausiSvyMagAccOrder[kk] <> 0 THEN
					a_bRcpLoaded[kk] := TRUE;
				END_IF
			END_FOR

		ELSE//Btm to top
			IF p_diRequestedMinSlt = 0 THEN
				p_diRequestedMinSlt := 1;
			END_IF

			FOR kk := 1 TO 3 DO//SIZEOF(a_tyCurrZ2Rcp)/SIZEOF(a_tyCurrZ2Rcp[1]) DO //btm to top
				//	rMinslt :=  p_diRequestedMinSlt + (a_tyCurrZ2Rcp[kk].rBottomClearanceHeight)/(p_diMagRcpCurrRcpSltToSlt/1000);
				IF ceil((a_tyCurrZ2Rcp[kk].rBottomClearanceHeight + p_diNtParamPullerHeightInMM )/(p_diMagRcpCurrRcpSltToSlt/1000)) >= p_diRequestedMinSlt THEN
					rMinslt :=  (a_tyCurrZ2Rcp[kk].rBottomClearanceHeight + p_diNtParamPullerHeightInMM )/(p_diMagRcpCurrRcpSltToSlt/1000) + 1;
				ELSE
					rMinslt :=  p_diRequestedMinSlt ;
				END_IF
				rMaxslt := p_diMagRcpCurrRcpTtlSlt - (a_tyCurrZ2Rcp[kk].rTopClearanceHeight + a_tyCurrZ2Rcp[kk].rThickness)/(p_diMagRcpCurrRcpSltToSlt/1000) + 1;
				rPitch := (a_tyCurrZ2Rcp[kk].rTopClearanceHeight + a_tyCurrZ2Rcp[kk].rBottomClearanceHeight + a_tyCurrZ2Rcp[kk].rThickness)/(p_diMagRcpCurrRcpSltToSlt/1000);
				IF rPitch = 0 THEN
					rPitch := 1;
				END_IF
				rNumInterval := (rMaxslt - rMinslt )/ceil(rPitch);
				diCalcedMin := REAL_TO_DINT(ceil(rMinslt)); //floor
				diCalcedPitch := REAL_TO_DINT(ceil(rPitch));
				diCalcedMax := REAL_TO_DINT((diCalcedMin + floor(rNumInterval)*ceil(rPitch)));

				IF diCalcedMax = p_diMagRcpCurrRcpTtlSlt + 1 THEN
					diCalcedMax := diCalcedMax - diCalcedPitch;
				END_IF
				//			IF diCalcedMin < p_diRequestedMinSlt THEN
				//				diModulus :=  p_diRequestedMinSlt/diCalcedMin;
				//				diCalcedMin := diCalcedMin + diModulus*diCalcedPitch;
				//			END_IF
				a_tyMagProps[kk].diMaxSlt := diCalcedMax;
				a_tyMagProps[kk].diMinSlt := diCalcedMin;
				a_tyMagProps[kk].diPitch  := diCalcedPitch;
				a_tyMagProps[kk].diWidth := REAL_TO_DINT(a_tyCurrZ2Rcp[kk].rWidth * 1000);
				IF a_tyCurrZ2Rcp[kk].sWorkOrderId <> '' AND diCalcedMin <> 0 AND p_ausiSvyMagAccOrder[kk] <> 0 THEN
					a_bRcpLoaded[kk] := TRUE;
				END_IF
			END_FOR

		END_IF

		bOverWriteMagProperties := FALSE;
	END_IF

	//Update and delete
	IF p_bOpsMagConvLD1ExtDelAutoRcp THEN
		memset(ADR(a_tyMagProps[1]),0,SIZEOF(a_tyMagProps[1]));
		memset(ADR(a_tyCurrZ2Rcp[1]),0,SIZEOF(a_tyCurrZ2Rcp[1]));
		p_ausiSvyMagAccOrder[1] := 0;  //bi-dir
		p_asSvyHermesMagGUID[1] := ''; //bi-dir
		a_bRcpLoaded[1] := FALSE;
	END_IF
	IF p_bOpsMagConvLD2ExtDelAutoRcp THEN
		memset(ADR(a_tyMagProps[2]),0,SIZEOF(a_tyMagProps[2]));
		memset(ADR(a_tyCurrZ2Rcp[2]),0,SIZEOF(a_tyCurrZ2Rcp[2]));
		p_ausiSvyMagAccOrder[2] := 0;
		p_asSvyHermesMagGUID[2] := '';
		a_bRcpLoaded[2] := FALSE;
	END_IF
	IF  p_bOpsMagConvLD3ExtDelAutoRcp THEN
		memset(ADR(a_tyMagProps[3]),0,SIZEOF(a_tyMagProps[3]));
		memset(ADR(a_tyCurrZ2Rcp[3]),0,SIZEOF(a_tyCurrZ2Rcp[3]));
		p_ausiSvyMagAccOrder[3] := 0;
		p_asSvyHermesMagGUID[3] := '';
		a_bRcpLoaded[3] := FALSE;
	END_IF

END_ACTION
```

#### PrecededBySelfInitial.st
```iecst
ACTION PrecededBySelfInitial:

	//Mag Detail
	fbFileRead1.sDevice			:= 'Retain';
	fbFileRead1.sFile			:= 'MagazineRcp';
	fbFileRead1.udiOffset		:= 0;
	fbFileRead1.p_Dest			:= ADR(a_tyCurrZ2Rcp);
	fbFileRead1.udiLen			:= SIZEOF(a_tyCurrZ2Rcp);
	fbFileRead1(bEn := FALSE);

	fbFileWrite1.sDevice	:= 'Retain';
	fbFileWrite1.sFile			:= 'MagazineRcp';
	fbFileWrite1.udiOffset		:= 0;
	fbFileWrite1.p_Src			:= ADR(a_tyZ2RcpWr);
	fbFileWrite1.udiLen			:= SIZEOF(a_tyZ2RcpWr);
	fbFileWrite1.udiOption		:= 0;
	fbFileWrite1(bEn := FALSE);

END_ACTION
```

#### PrecededBySelfLink.st
```iecst
ACTION PrecededBySelfLink:

	//For Accepting BA or BF from HermesA/B
//	p_bHermesBADataAccepted := p_bHermesABAAccepted OR p_bHermesBBAAccepted;
//	IF p_bHermesABAAccepted THEN
//		p_tyHermesBARcv ACCESS p_USHermesABoardAvailableRcv;
//	ELSIF  p_bHermesBBAAccepted THEN
//		p_tyHermesBARcv ACCESS p_USHermesABoardAvailableRcv;
//	END_IF

//	p_bHermesBFDataAccepted	:= 	p_bHermesABFAccepted OR p_bHermesBBFAccepted;
//	IF p_bHermesABFAccepted THEN
//		p_tyHermesBFRcv ACCESS p_USHermesABoardForecastRcv;
//	ELSIF p_bHermesBBFAccepted THEN
//		p_tyHermesBFRcv ACCESS p_USHermesBBoardForecastRcv;
//	END_IF

	//LCS Data ....

	//Z1 Accepting Condition
	p_bZ1AccNewRcpCondition := (p_bLinkOpsRun = TRUE) AND (p_bLinkOpsTravLifLDInitDone = TRUE) AND (p_bLinkPshrConvHvBrd = FALSE);

	//Z2 Accepting Condition
	p_bZ2AccNewRcpCondition := (p_bLinkOpsRun = TRUE) AND (p_bLinkOpsMagConvLD1InitDone AND p_bLinkOpsMagConvLD2InitDone AND p_bLinkOpsMagConvLD3InitDone);

END_ACTION
```

#### Package Logical/AutoRcp/AutoRcp/PrecededByF1 - Intended for F2 only

#### PrecededByF1Background1.st
```iecst
ACTION PrecededByF1Background1:
	//Requesting
//	tyCurrReqMagRcp.diMaxSltValue := p_tyInternalReqProdRcp.diMaxSltValue;
//	tyCurrReqMagRcp.diMinSltValue := p_tyInternalReqProdRcp.diMinSltValue;
//	tyCurrReqMagRcp.diPitch  := p_tyInternalReqProdRcp.diPitch;
//	tyCurrReqMagRcp.diWidthInUM  := p_tyInternalReqProdRcp.diWidthInUM;
//	tyCurrReqMagRcp.sRcpNm   := p_tyInternalReqProdRcp.sRcpNm;
	memcpy(ADR(tyCurrReqMagRcp) , ADR(p_tyInternalReqProdRcp) , SIZEOF(tyCurrReqMagRcp));

	IF eStatus = Error THEN
		p_ausiLCSLFMagAccOrder[p_usiLCSLFMagOrderPos] := 0;  //bi-dir
		IF p_usiLCSLFMagOrderPos = 1 THEN
			p_bLinkOpsMagConvLD1QueryWO := FALSE; //bi-dir ,cancel bQueryWO
		ELSIF p_usiLCSLFMagOrderPos =2 THEN
			p_bLinkOpsMagConvLD2QueryWO := FALSE; //bi-dir
		ELSIF p_usiLCSLFMagOrderPos =3 THEN
			p_bLinkOpsMagConvLD3QueryWO := FALSE; //bi-dir
		END_IF
		p_usiLCSLFMagOrderPos := 0;	  //bi-dir
	END_IF

	//For Zone 1 Initialization Only (follow internal rcp width)
	IF bInitializedFollower1Done = FALSE THEN
		IF p_tyInternalReqProdRcp.diWidthInUM <> 0 THEN
			diTravLifWidth := p_tyInternalReqProdRcp.diWidthInUM; //Z1Rcp == TravLif
			bOverWriteTravLifProperties := TRUE;
			bInitializedFollower1Done := TRUE;
		END_IF
	END_IF

	IF p_usiLCSLFMagOrderPos > 0 AND eStatus <> Error THEN
		a_tyAutoRcpInternal[p_usiLCSLFMagOrderPos] := tyCurrReqMagRcp;
		//updare min max pitch to buffer
		a_tyMagProps[p_usiLCSLFMagOrderPos].diMinSlt := tyCurrReqMagRcp.diMinSltValue;
		a_tyMagProps[p_usiLCSLFMagOrderPos].diMaxSlt := tyCurrReqMagRcp.diMaxSltValue;
		a_tyMagProps[p_usiLCSLFMagOrderPos].diPitch := tyCurrReqMagRcp.diPitch;

		bOverWriteMagProperties := TRUE;
		usiChg := usiChg + 1;
		p_usiLCSLFMagOrderPos := 0;	  //bi-dir
	END_IF

	//Follower1 //Changed to a_tyCurrZ2Rcp //Assign when received WO and empty rcp
	FOR usi := 1 TO 3 DO
		IF p_ausiLCSLFMagAccOrder[usi] = 10 AND eStatus <> Error THEN
			IF memcmp(ADR(a_tyAutoRcpInternal[usi]) , ADR(a_tyAutoRcpFollower1) , SIZEOF(a_tyAutoRcpInternal[usi])) <> 0 THEN
				bTravLifWidthDiffBlk := TRUE; //block travlif USallow
				IF p_bZ1AccNewRcpCondition THEN
					a_tyAutoRcpFollower1 := a_tyAutoRcpInternal[usi]; //output to follower 1
					a_bRcpLoaded[usi] := TRUE;
				END_IF
			ELSE
				bTravLifWidthDiffBlk := FALSE;
			END_IF
		END_IF
	END_FOR

	//Convert to Width for F1 //Changed to a_tyCurrZ2Rcp
	IF p_ausiLCSLFMagAccOrder[1] = 0 AND p_ausiLCSLFMagAccOrder[2] = 0 AND p_ausiLCSLFMagAccOrder[3] = 0 THEN
		diTravLifWidth := 100000;
	ELSE
		FOR usi := 1 TO 3 DO
			IF p_ausiLCSLFMagAccOrder[usi] = 10 AND p_bConvHvBrd = FALSE THEN
				a_tyAutoRcpFollower1 := a_tyAutoRcpInternal[usi];
				diTravLifPitch := a_tyAutoRcpInternal[usi].diPitch;
				diTravLifWidth := a_tyAutoRcpInternal[usi].diWidthInUM ;
				EXIT;
				//diTravLifWidth := REAL_TO_DINT(a_tyCurrZ2Rcp[usi].rWidth*1000);
			END_IF
		END_FOR
	END_IF

	//Update and delete
	IF p_bOpsMagConvLD1ExtDelAutoRcp THEN
		p_ausiLCSLFMagAccOrder[1] := 0;  //bi-dir
		a_bRcpLoaded[1] := FALSE;
	END_IF
	IF p_bOpsMagConvLD2ExtDelAutoRcp THEN
		p_ausiLCSLFMagAccOrder[2] := 0;
		a_bRcpLoaded[2] := FALSE;
	END_IF
	IF  p_bOpsMagConvLD3ExtDelAutoRcp THEN
		p_ausiLCSLFMagAccOrder[3] := 0;
		a_bRcpLoaded[3] := FALSE;
	END_IF

END_ACTION
```

#### PrecededByF1Initial.st
```iecst
ACTION PrecededByF1Initial:

	//Mag Detail (Rcp)
	fbFileRead1.sDevice			:= 'Retain';
	fbFileRead1.sFile			:= 'MagazinePropsRcp';
	fbFileRead1.udiOffset		:= 0;
	fbFileRead1.p_Dest			:= ADR(a_tyAutoRcpInternal);
	fbFileRead1.udiLen			:= SIZEOF(a_tyAutoRcpInternal);
	fbFileRead1(bEn := FALSE);

	fbFileWrite1.sDevice	:= 'Retain';
	fbFileWrite1.sFile			:= 'MagazinePropsRcp';
	fbFileWrite1.udiOffset		:= 0;
	fbFileWrite1.p_Src			:= ADR(a_tyAutoRcpInternalWr);
	fbFileWrite1.udiLen			:= SIZEOF(a_tyAutoRcpInternalWr);
	fbFileWrite1.udiOption		:= 0;
	fbFileWrite1(bEn := FALSE);

END_ACTION
```

#### PrecededByF1Link.st
```iecst
ACTION PrecededByF1Link:

	//Z1 Accepting Condition
	p_bZ1AccNewRcpCondition := (p_bLinkOpsRun = TRUE) AND (p_bLinkOpsTravLifLDInitDone = TRUE) AND (p_bLinkPshrConvHvBrd = FALSE);

	//Z2 Accepting Condition
	p_bZ2AccNewRcpCondition := (p_bLinkOpsRun = TRUE) AND (p_bLinkOpsMagConvLD1InitDone AND p_bLinkOpsMagConvLD2InitDone AND p_bLinkOpsMagConvLD3InitDone);

END_ACTION
```

#### Act_InitGlobal.st - Change By Project
```iecst
(** 2019-06-12 **)
ACTION Act_InitGlobal:

	(* Always Change If Project Change *)

	//Pass Data To Link
	p_bLinkStartupRun ACCESS p_StartupRun;

	p_bLinkOpsRun ACCESS p_OpsRun;
	p_eLinkNtParamProjMag ACCESS p_NtParamProjMag;
	p_tyNtParamAutoRcpParamLmt ACCESS p_NtParamAutoRcpParamLmt;
	p_diNtParamProdRcpMaxWidth ACCESS p_NtParamProdRcpMaxWidth;
	p_diNtParamProdRcpMinWidth ACCESS p_NtParamProdRcpMinWidth;
	p_tySendWorkOrderData ACCESS p_SvyHermesSendWorkOrderData;
	p_bSndWorkOrderInfo ACCESS p_SndWorkOrderInfo;
	p_ausiSvyMagAccOrder ACCESS p_SvyHermesMagAccOrder;
	p_asSvyHermesMagGUID ACCESS p_SvyHermesMagGUID;
	p_usiSvyMagOrderPos ACCESS p_SvyHermesMagOrderPos;

	p_bLinkOpsMagConvLD1QueryWO ACCESS p_OpsMagConvLD1QueryWO;
	p_bLinkOpsMagConvLD2QueryWO ACCESS p_OpsMagConvLD2QueryWO;
	p_bLinkOpsMagConvLD3QueryWO ACCESS p_OpsMagConvLD3QueryWO;

	//Pass Data To Internal Use
	p_udiRstErr ACCESS p_RstErrReset;
//	p_tyInternalReqProdRcp ACCESS p_Follower1UpdtProdRcp;	//Follower 2 Assign With Follower 1 Recipe
//	p_sProgNm ACCESS p_NtParamFollower2ProgNm;
	p_bNtSettingsLoadDone ACCESS p_StartupNtSettingsLoadDone;

	p_bPrep ACCESS p_NtParamAutoRcpPrep;
	p_diNtParamPullerHeightInMM ACCESS p_NtParamPullerHeightInMM;
	//Zone 1
	p_bLinkPshrConvHvBrd ACCESS p_PullConvHvBrd;
	p_bLinkOpsTravLifLDInitDone ACCESS p_OpsTravLifLDInitDone;

	//Zone 2
	p_bLinkOpsMagConvLD1InitDone ACCESS p_OpsMagConvLD1InitDone;
	p_bLinkOpsMagConvLD2InitDone ACCESS p_OpsMagConvLD2InitDone;
	p_bLinkOpsMagConvLD3InitDone ACCESS p_OpsMagConvLD3InitDone;
	p_udiOpsMagConvLD1MagAllwGo ACCESS p_OpsMagConvLD1MagAllwGo;
	p_udiOpsMagConvLD2MagAllwGo ACCESS p_OpsMagConvLD2MagAllwGo;
	p_udiOpsMagConvLD3MagAllwGo ACCESS p_OpsMagConvLD3MagAllwGo;

	p_bOpsMagConvLD1ExtDelAutoRcp ACCESS p_OpsMagConvLD1ExtDelAutoRcp;
	p_bOpsMagConvLD2ExtDelAutoRcp ACCESS p_OpsMagConvLD2ExtDelAutoRcp;
	p_bOpsMagConvLD3ExtDelAutoRcp ACCESS p_OpsMagConvLD3ExtDelAutoRcp;

	p_bBuffer1MagPresent ACCESS p_Buffer1MagPresent;
	p_bBuffer2MagPresent ACCESS p_Buffer2MagPresent;
	p_bBuffer3MagPresent ACCESS p_Buffer3MagPresent;

	p_bBuffer1MagRemoved ACCESS p_Buffer1MagPresent;
	p_bBuffer2MagRemoved ACCESS p_Buffer2MagPresent;
	p_bBuffer3MagRemoved ACCESS p_Buffer3MagPresent;

	p_tyBuffer1BffrStat ACCESS p_Buffer1BffrStat ;
	p_tyBuffer2BffrStat ACCESS p_Buffer2BffrStat ;
	p_tyBuffer3BffrStat ACCESS p_Buffer3BffrStat ;

//	p_bMagAW1WidthDiff ACCESS p_MagAWOpen1WidthPosDiff;
//	p_bMagAW2WidthDiff ACCESS p_MagAWOpen2WidthPosDiff;
//	p_bMagAW3WidthDiff ACCESS p_MagAWOpen3WidthPosDiff;

	//Hermes A accepted the BA
//	p_bHermesABAAccepted ACCESS p_USHermesABAAccepted; //brd avail
//	p_bHermesABFAccepted ACCESS p_USHermesABFAccepted; //brd forecast

	//Hermes B accepeted the BA
//	p_bHermesBBAAccepted ACCESS p_USHermesBBAAccepted;
//	p_bHermesBBFAccepted ACCESS p_USHermesBBFAccepted;

	p_diMagRcpCurrRcpTtlSlt ACCESS p_MagRcpCurrRcpTtlSlt;
	p_diMagRcpCurrRcpSltToSlt ACCESS p_MagRcpCurrRcpSltToSlt;

//	p_tyInternalReqProdRcp ACCESS p_ProdRcpCurrRcp0;
	p_bProdSelTopToBtm ACCESS p_ProdRcpCurrRcp1TopToBtm;

	p_bConvHvBrd ACCESS p_PullConvHvBrd;

	//We Fab
	p_tyInternalReqProdRcp ACCESS p_ProdRcpCurrRcp0;	//Follower 0
	p_eNtParamAutoRcpPrecededBy ACCESS p_NtParamAutoRcpPrecededBy;
	p_ausiLCSLFMagAccOrder ACCESS p_LCSLFMagAccOrder;
	p_usiLCSLFMagOrderPos ACCESS p_LCSLFMagOrderPos;

END_ACTION
```

#### InputRef_Link.var - Change By Project
```iecst
(*2019-05-07*)
(**)
VAR
	p_bLinkStartupRun : REFERENCE TO BOOL;
END_VAR
(**)
VAR
	p_bLinkOpsRun : REFERENCE TO BOOL;
	p_eLinkNtParamProjMag : REFERENCE TO eLDMag;
	p_tyNtParamAutoRcpParamLmt : REFERENCE TO AutoRcpLmt;
	p_diNtParamProdRcpMaxWidth : REFERENCE TO DINT;
	p_diNtParamProdRcpMinWidth : REFERENCE TO DINT;
	p_diNtParamPullerHeightInMM : REFERENCE TO DINT;
	p_bLinkPshrConvHvBrd : REFERENCE TO BOOL;
	p_bLinkOpsTravLifLDInitDone : REFERENCE TO BOOL;
	p_bLinkMagConvInitDone : BOOL;
	p_bLinkNtParamProjMagConv1Prep : REFERENCE TO BOOL;
	p_bLinkNtParamProjMagConv2Prep : REFERENCE TO BOOL;
	p_bLinkNtParamProjMagConv3Prep : REFERENCE TO BOOL;
	p_bLinkBffr1MagRemoved : REFERENCE TO BOOL;
	p_bLinkBffr2MagRemoved : REFERENCE TO BOOL;
	p_bLinkBffr3MagRemoved : REFERENCE TO BOOL;
	p_bLinkOpsMagUL1InitDone : REFERENCE TO BOOL;
	p_bLinkOpsMagUL2InitDone : REFERENCE TO BOOL;
	p_bLinkOpsMagUL3InitDone : REFERENCE TO BOOL;
	p_bLinkOpsMagConvLD1InitDone : REFERENCE TO BOOL;
	p_bLinkOpsMagConvLD2InitDone : REFERENCE TO BOOL;
	p_bLinkOpsMagConvLD3InitDone : REFERENCE TO BOOL;
	p_tyBuffer1BffrStat : REFERENCE TO tyBffrStat;
	p_tyBuffer2BffrStat : REFERENCE TO tyBffrStat;
	p_tyBuffer3BffrStat : REFERENCE TO tyBffrStat;
	p_bMagAW1WidthDiff : REFERENCE TO BOOL;
	p_bMagAW2WidthDiff : REFERENCE TO BOOL;
	p_bMagAW3WidthDiff : REFERENCE TO BOOL;
	p_udiOpsMagConvLD1MagAllwGo : REFERENCE TO UDINT;
	p_udiOpsMagConvLD2MagAllwGo : REFERENCE TO UDINT;
	p_udiOpsMagConvLD3MagAllwGo : REFERENCE TO UDINT;
	p_bOpsMagConvLD1ExtDelAutoRcp : REFERENCE TO BOOL;
	p_bOpsMagConvLD2ExtDelAutoRcp : REFERENCE TO BOOL;
	p_bOpsMagConvLD3ExtDelAutoRcp : REFERENCE TO BOOL;
	p_bZ1AccNewRcpCondition : REFERENCE TO BOOL;
	p_bZ2AccNewRcpCondition : REFERENCE TO BOOL;
	p_diRequestedMinSlt : REFERENCE TO DINT;
	p_bHermesBADataAccepted : REFERENCE TO BOOL;
	p_bHermesBFDataAccepted : REFERENCE TO BOOL;
	p_bHermesBBAAccepted : REFERENCE TO BOOL;
	p_bHermesABAAccepted : REFERENCE TO BOOL;
	p_bHermesBBFAccepted : REFERENCE TO BOOL;
	p_bHermesABFAccepted : REFERENCE TO BOOL;
	p_tyHermesBARcv : REFERENCE TO tyHermesBoardAvailable;
	p_tyHermesBFRcv : REFERENCE TO tyHermesBoardForecast;
	p_diMagRcpCurrRcpSltToSlt : REFERENCE TO DINT;
	p_diMagRcpCurrRcpTtlSlt : REFERENCE TO DINT;
	p_bBuffer1MagPresent : REFERENCE TO BOOL;
	p_bBuffer2MagPresent : REFERENCE TO BOOL;
	p_bBuffer3MagPresent : REFERENCE TO BOOL;
	p_bBuffer1MagRemoved : REFERENCE TO BOOL;
	p_bBuffer2MagRemoved : REFERENCE TO BOOL;
	p_bBuffer3MagRemoved : REFERENCE TO BOOL;
END_VAR
(**)
VAR
	bOpsInitDone : BOOL;
	p_eLinkUIProdRcpAct : REFERENCE TO eProdRcpAction;
	p_eProdRcpStat : REFERENCE TO eProdRcpAction;
	p_eProdRcpStatus : REFERENCE TO eFBStatus;
	p_tyProdRcpCurrRcpWr : REFERENCE TO tyProdRcpParam;
	p_tySendWorkOrderData : REFERENCE TO tyHermesSendWorkOrderInfo;
	p_bSndWorkOrderInfo : REFERENCE TO BOOL;
	p_ausiSvyMagAccOrder : REFERENCE TO ARRAY[1..3] OF USINT;
	p_asSvyHermesMagGUID : REFERENCE TO ARRAY[1..3] OF STRING[80];
	p_usiSvyMagOrderPos : REFERENCE TO USINT;
	p_bLinkOpsMagConvLD1QueryWO : REFERENCE TO BOOL;
	p_bLinkOpsMagConvLD2QueryWO : REFERENCE TO BOOL;
	p_bLinkOpsMagConvLD3QueryWO : REFERENCE TO BOOL;
END_VAR
(*WeFab*)
VAR
	p_ausiLCSLFMagAccOrder : REFERENCE TO ARRAY[1..3] OF USINT;
	p_usiLCSLFMagOrderPos : REFERENCE TO USINT;
END_VAR
```

#### Act_LinkEn.st - Change By Project
```iecst
(** 2019-04-26 **)
ACTION Act_LinkEn:

	//Link bPrep, bEn & bDis
	//p_bDis	:= (p_bLinkStartupRun = TRUE);
	//p_bPrep	:= p_bNtParamAutoRcpPrep;

END_ACTION
```

#### Act_Link.st - Change By Project
```iecst
(** 2019-07-04 **)
ACTION Act_Link:

	CASE p_eNtParamAutoRcpPrecededBy OF
		PrecededBySelf:
			PrecededBySelfLink;
		PrecededByF1:
			PrecededByF1Link;
	END_CASE

	//for comparing Rcp
	a_tyBffrStat[1] := p_tyBuffer1BffrStat;
	a_tyBffrStat[2] := p_tyBuffer2BffrStat;
	a_tyBffrStat[3] := p_tyBuffer3BffrStat;

	a_udiMagAllwGo[1] := p_udiOpsMagConvLD1MagAllwGo;
	a_udiMagAllwGo[2] := p_udiOpsMagConvLD2MagAllwGo;
	a_udiMagAllwGo[3] := p_udiOpsMagConvLD3MagAllwGo;

	a_bBufferMagPresent[1] := p_bBuffer1MagPresent;
	a_bBufferMagPresent[2] := p_bBuffer2MagPresent;
	a_bBufferMagPresent[3] := p_bBuffer3MagPresent;

	//	a_bMagAWWidthDiff[1] := p_bMagAW1WidthDiff;
	//	a_bMagAWWidthDiff[2] := p_bMagAW2WidthDiff;
	//	a_bMagAWWidthDiff[3] := p_bMagAW3WidthDiff;

	//pa_bInternalReqProdRcpDiff[ii]

	//p_bUpdtProdRcpDiff			:= memcmp(ADR(p_tyCurrProdRcp) , ADR(tyUpdtProdRcp) , SIZEOF(p_tyCurrProdRcp)) <> 0;

END_ACTION
```

#### Cyclic.st - Do Not Change!!!
```iecst
(** 2019-04-21 **)
PROGRAM _CYCLIC

	IF bInitDone = FALSE THEN
		bInitDone	:= TRUE;

		Act_InitLocal;
		Act_InitGlobal;

	ELSIF bInitialDone = FALSE THEN
		IF p_bNtSettingsLoadDone = TRUE THEN
			bInitialDone	:= TRUE;

			Act_Initial;
		END_IF

	ELSE

		Act_RstErr;
		Act_LinkAction;
		Act_Action;
	//	Act_LinkEn;

		IF (p_bPrep = TRUE) AND (p_bEn = TRUE) AND (p_bDis = FALSE) THEN
			Act_Link;
			Act_Main;
			Act_Background;
			Act_Background2;
		ELSE
			Act_Main_Disable;

		END_IF

		Act_Alarm;

	END_IF

END_PROGRAM
```

#### Act_InitLocal.st - Do Not Change!!!
```iecst
(** 2020-08-06 **)
ACTION Act_InitLocal:

	//Input Reference Link To Local Variable
	p_udiRstErr ACCESS ADR(udiRstErr);
	p_bPrep ACCESS ADR(bPrep);
	p_bEn ACCESS ADR(bEn);
	p_bDis ACCESS ADR(bDis);
	p_sIPAddr ACCESS ADR(sIPAddr);
	p_sMcNm ACCESS ADR(sMcNm);
	p_bAWPrep ACCESS ADR(bAWPrep);
	p_bAWDis ACCESS ADR(bAWDis);
	p_bMnlAccData ACCESS ADR(bMnlAccData);
	p_bSectionLeader ACCESS ADR(bSectionLeader);
	p_sMagRcpNm ACCESS ADR(sMagRcpNm);
	p_diWidthLimit ACCESS ADR(diWidthLimit);
	p_bUSWidthChkPrep ACCESS ADR(bUSWidthChkPrep);
	p_bUSWidthChkEn ACCESS ADR(bUSWidthChkEn);
	p_bUSWidthChkSen ACCESS ADR(bUSWidthChkSen);
	p_bDSWidthChkPrep ACCESS ADR(bDSWidthChkPrep);
	p_bDSWidthChkEn ACCESS ADR(bDSWidthChkEn);
	p_bDSWidthChkSen ACCESS ADR(bDSWidthChkSen);
	p_bProdWidthChk ACCESS ADR(bProdWidthChk);
	p_bUIProdAccData ACCESS ADR(bUIProdAccData);
	p_bUIProdUpdtData ACCESS ADR(bUIProdUpdtData);
	p_bUIMagAccData ACCESS ADR(bUIMagAccData);

	p_tyCmpRcp ACCESS ADR(tyCurrProdRcp);
	p_sCurrMagRcpNm ACCESS ADR(sCurrMagRcpNm);
	p_eTimeStat ACCESS ADR(eTimeStat);
	p_eTimeStatus ACCESS ADR(eTimeStatus);
	p_bAccNewRcpCond ACCESS ADR(bAccNewRcpCond);
	p_bUpdtNewRcpCond ACCESS ADR(bUpdtNewRcpCond);
	p_bAutoUpdtData ACCESS ADR(bAutoUpdtData);
	p_sInfoMsg ACCESS ADR(sInfoMsg);
	p_bInternalUse ACCESS ADR(bInternalUse);
	p_tyInternalReqProdRcp ACCESS ADR(tyInternalReqProdRcp);
	p_bNewBrdEnteredCond ACCESS ADR(bNewBrdEnteredCond);
	p_bOldBrdExitedCond ACCESS ADR(bOldBrdExitedCond);
	p_bRlsBrd ACCESS ADR(bRlsBrd);
	p_tyToLeaderProdRcp ACCESS ADR(tyToLeaderProdRcp);
	pa_bInternalReqProdRcpDiff ACCESS ADR(a_bInternalReqProdRcpDiff);
	p_bUpdtProdRcpDiff ACCESS ADR(bUpdtProdRcpDiff);
	p_bRlsBrdProdRcpDiff ACCESS ADR(bRlsBrdProdRcpDiff);
	p_sProgNm ACCESS ADR(sProgNm);
	p_bNtSettingsLoadDone ACCESS ADR(bNtSettingsLoadDone);
	p_tOnlineChkDlyTm ACCESS ADR(tOnlineChkDlyTm);
	p_bManual ACCESS ADR(bManual);
	p_bErr ACCESS ADR(bErr);
	p_bWarning ACCESS ADR(bWarning);
	p_bOps ACCESS ADR(bOps);
	p_bStandby ACCESS ADR(bStandby);
	p_eAWStat ACCESS ADR(eAWStat);
	p_bWidth2Prep ACCESS ADR(bWidth2Prep);
	p_tyProdRcpCurrRcpWr ACCESS ADR(bDBAOnWOAlign);
	p_eLinkUIProdRcpAct ACCESS ADR(bDBAOnWOAlign);

	p_bZ1AccNewRcpCondition ACCESS ADR(bZ1AccNewRcpCondition);
	p_bZ2AccNewRcpCondition ACCESS ADR(bZ2AccNewRcpCondition);
	p_tyHermesBARcv ACCESS ADR(tyHermesBAAccpt);
	p_tyHermesBFRcv ACCESS ADR(tyHermesBFAccpt);
	p_bHermesBADataAccepted ACCESS  ADR(bHermesBAAccpt);
	p_bHermesBFDataAccepted ACCESS  ADR(bHermesBFAccpt);
	p_diRequestedMinSlt ACCESS ADR(diRequestedMinSlt);
END_ACTION
```

#### Act_Initial.st - Do Not Change!!!
```iecst
(** 2020-08-06 **)
ACTION Act_Initial:
	fbDirCreate1.sDevice	:= 'F';
	fbDirCreate1.sDirName	:= 'User';
	fbDirCreate1(bEn := FALSE);

	fbDirCreate2.sDevice	:= 'User';
	fbDirCreate2.sDirName	:= 'Retain';
	fbDirCreate2(bEn := FALSE);

	CASE p_eNtParamAutoRcpPrecededBy OF
		PrecededBySelf:
			PrecededBySelfInitial;
		PrecededByF1:
			PrecededByF1Initial;
	END_CASE

END_ACTION
```

#### Act_Background.st - Do Not Change!!!
```iecst
(** 2021-05-18 **)
ACTION Act_Background:

	CASE p_eNtParamAutoRcpPrecededBy OF
		PrecededBySelf:
			PrecededBySelfBackground1;
		PrecededByF1:
			PrecededByF1Background1;
	END_CASE

	//if different, write one time
	IF usiPrevChg <> usiChg
		AND (eStatus = Idle AND eStat = AutoRcpActIdle)  THEN
		IF p_eNtParamAutoRcpPrecededBy = 0 THEN
			a_tyZ2RcpWr := a_tyCurrZ2Rcp;
		ELSIF p_eNtParamAutoRcpPrecededBy = 1 THEN
			a_tyAutoRcpInternalWr := a_tyAutoRcpInternal;
		END_IF
		p_eAct := AutoRcpActWriteRetain;
	END_IF
	IF eStatus = Done AND eStat = AutoRcpActWriteRetain THEN
		usiPrevChg :=  usiChg;
		p_eAct := AutoRcpActIdle;
	END_IF

END_ACTION
```

#### Act_Background2.st - Do Not Change!!!
```iecst
(** 2021-05-18 **)
ACTION Act_Background2:

	CASE p_eNtParamAutoRcpPrecededBy OF
		PrecededBySelf:
			PrecededBySelfBackground2;
		PrecededByF1:
			PrecededByF1Background2;
	END_CASE

END_ACTION
```

#### Act_Main.st - Do Not Change!!!
```iecst
(** 2021-08-01 **)
ACTION Act_Main:

	IF eStatOld <> eStat THEN
		fbDirCreate1(bEn := FALSE);
		fbDirCreate2(bEn := FALSE);

		fbFileRead1(bEn := FALSE);
		fbFileWrite1(bEn := FALSE);

		usiStep			:= 0;
		bFileNotFound	:= FALSE;

		//sStatTxt	:= a_sStatText[eStat];

		eStatOld	:= eStat;

		eStatus		:= Busy;
	END_IF

	//Main
	CASE eStat OF

		AutoRcpActIdle:
			eStatus	:= Idle;

		AutoRcpActCreateDir:
			IF eStatus = Idle OR eStatus = Busy THEN

				eStatus	:= Busy;

				CASE usiStep OF
					0:
						fbDirCreate1(bEn := TRUE);
						IF fbDirCreate1.udiStatus = 0 THEN
							usiStep	:= 1;
						ELSIF fbDirCreate1.udiStatus < 65534 THEN
							eStatus		:= Error;

							IF fbDirCreate1.udiStatus = 1908 THEN
								udiStatus	:= 10000;	//Create User Directory Error
							ELSE
								udiStatus	:= fbDirCreate1.udiStatus;
							END_IF
						END_IF

					1:
						fbDirCreate2(bEn := TRUE);
						IF fbDirCreate2.udiStatus = 0 THEN
							eStatus	:= Done;
						ELSIF fbDirCreate2.udiStatus < 65534 THEN
							eStatus		:= Error;

							IF fbDirCreate2.udiStatus = 1908 THEN
								udiStatus	:= 10001;	//Create Retain Directory Error
							ELSE
								udiStatus	:= fbDirCreate2.udiStatus;
							END_IF
						END_IF

				END_CASE

			END_IF

		AutoRcpActReadRetain:
			IF eStatus = Idle OR eStatus = Busy THEN

				eStatus	:= Busy;

//				fbFileRead1.p_Dest	:= p_udiRetainDataAddr1;
//				fbFileRead1.udiLen	:= p_udiRetainDataLen1;
				fbFileRead1(bEn := TRUE);

				IF fbFileRead1.udiStatus = 0 THEN
					eStatus	:= Done;
					a_tyZ2RcpWr := a_tyCurrZ2Rcp;
					bOverWriteMagProperties := TRUE;
					bOverWriteTravLifProperties := TRUE;
				ELSIF fbFileRead1.udiStatus < 65534 THEN
					eStatus	:= Error;

					IF fbFileRead1.udiStatus = 1900 THEN
						udiStatus	:= 10002;	//File Open Error While Reading Retain File
					ELSIF fbFileRead1.udiStatus = 1902 THEN
						udiStatus	:= 10003;	//File Read Error While Reading Retain File
					ELSIF fbFileRead1.udiStatus = 1904 THEN
						udiStatus	:= 10004;	//File Close Error While Reading Retain File
					ELSIF fbFileRead1.udiStatus = 1915 THEN
						eStatus			:= Done;
						bFileNotFound	:= TRUE;
					ELSE
						udiStatus	:= fbFileRead1.udiStatus;
					END_IF
				END_IF

			END_IF

		AutoRcpActWriteRetain:
			IF eStatus = Idle OR eStatus = Busy THEN

				eStatus	:= Busy;

//				fbFileWrite1.p_Src	:= p_udiRetainDataAddr1;
//				fbFileWrite1.udiLen	:= p_udiRetainDataLen1;
				fbFileWrite1(bEn := TRUE);

				IF fbFileWrite1.udiStatus = 0 THEN
					eStatus	:= Done;
				ELSIF fbFileWrite1.udiStatus < 65534 THEN
					eStatus	:= Error;

					IF fbFileWrite1.udiStatus = 1900 THEN
						udiStatus	:= 10005;	//File Open Error While Writing Retain File
					ELSIF fbFileWrite1.udiStatus = 1901 THEN
						udiStatus	:= 10006;	//File Create Error While Writing Retain File
					ELSIF fbFileWrite1.udiStatus = 1903 THEN
						udiStatus	:= 10007;	//File Write Error While Writing Retain File
					ELSIF fbFileWrite1.udiStatus = 1904 THEN
						udiStatus	:= 10008;	//File Close Error While Writing Retain File
					ELSIF fbFileWrite1.udiStatus = 1914 THEN
						udiStatus	:= 10009;	//Directory Does Not Exist While Writing Retain File
					ELSE
						udiStatus	:= fbFileWrite1.udiStatus;
					END_IF
				END_IF

			END_IF

		ELSE
			IF eStatus = Idle OR eStatus = Busy THEN
				eStatus	:= Done;
			END_IF

	END_CASE

END_ACTION
```

#### InputRef.var - Do Not Change!!!
```iecst
(*2020-08-06*)
(**)
(*General*)
VAR
	p_eAct : REFERENCE TO eAutoRcpAction;
	p_udiRstErr : REFERENCE TO UDINT;
	p_bPrep : REFERENCE TO BOOL;
	p_bEn : REFERENCE TO BOOL;
	p_bDis : REFERENCE TO BOOL;
END_VAR
(**)
(*Configuration*)
VAR
	p_eAWStat : REFERENCE TO eAWAction;
	p_sIPAddr : REFERENCE TO STRING[15];
END_VAR
(**)
(*Input*)
VAR
	p_sMcNm : REFERENCE TO STRING[30];
	p_bAWPrep : REFERENCE TO BOOL;
	p_bAWDis : REFERENCE TO BOOL;
	p_bMnlAccData : REFERENCE TO BOOL;
	p_bSectionLeader : REFERENCE TO BOOL;
	p_sMagRcpNm : REFERENCE TO STRING[30];
	p_diWidthLimit : REFERENCE TO DINT;
	p_bWidth2Prep : REFERENCE TO BOOL;
	p_bUSWidthChkPrep : REFERENCE TO BOOL;
	p_bUSWidthChkEn : REFERENCE TO BOOL;
	p_bUSWidthChkSen : REFERENCE TO BOOL;
	p_bDSWidthChkPrep : REFERENCE TO BOOL;
	p_bDSWidthChkEn : REFERENCE TO BOOL;
	p_bDSWidthChkSen : REFERENCE TO BOOL;
	p_bProdWidthChk : REFERENCE TO BOOL;
	p_bUIProdAccData : REFERENCE TO BOOL;
	p_bUIProdUpdtData : REFERENCE TO BOOL;
	p_bUIMagAccData : REFERENCE TO BOOL;
	p_tyCmpRcp : REFERENCE TO tyBoardProperty;
	p_sCurrMagRcpNm : REFERENCE TO STRING[30];
	p_eTimeStat : REFERENCE TO eTimeAction;
	p_eTimeStatus : REFERENCE TO eFBStatus;
	p_bAccNewRcpCond : REFERENCE TO BOOL;
	p_bUpdtNewRcpCond : REFERENCE TO BOOL;
	p_bAutoUpdtData : REFERENCE TO BOOL;
	p_sInfoMsg : REFERENCE TO STRING[200];
	p_bInternalUse : REFERENCE TO BOOL;
	p_tyInternalReqProdRcp : REFERENCE TO tyProdRcpParam;
	p_bNewBrdEnteredCond : REFERENCE TO BOOL;
	p_bOldBrdExitedCond : REFERENCE TO BOOL;
	p_bRlsBrd : REFERENCE TO BOOL;
	p_tyToLeaderProdRcp : REFERENCE TO tyProdRcpParam;
	pa_bInternalReqProdRcpDiff : REFERENCE TO ARRAY[0..3] OF BOOL;
	p_bUpdtProdRcpDiff : REFERENCE TO BOOL;
	p_bRlsBrdProdRcpDiff : REFERENCE TO BOOL;
	p_sProgNm : REFERENCE TO STRING[15];
	p_bNtSettingsLoadDone : REFERENCE TO BOOL;
	p_tOnlineChkDlyTm : REFERENCE TO TIME;
	p_bManual : REFERENCE TO BOOL;
	p_bErr : REFERENCE TO BOOL;
	p_bWarning : REFERENCE TO BOOL;
	p_bOps : REFERENCE TO BOOL;
	p_bStandby : REFERENCE TO BOOL;
	p_bProdSelTopToBtm : REFERENCE TO BOOL;
	p_bConvHvBrd : REFERENCE TO BOOL;
	p_eNtParamAutoRcpPrecededBy : REFERENCE TO eAutoRcpPreceded;
END_VAR
```

#### Local.var - Do Not Change!!!
```iecst
(*2021-05-18*)
(**)
(*Local Action, State & Status*)
VAR
	eAct : eAutoRcpAction;
	eStatus : eFBStatus := Idle;
	udiStatus : UDINT := 0;
	eStatOld : eAutoRcpAction := AutoRcpActIdle;
	eStat : eAutoRcpAction;
	usiStep : USINT;
END_VAR
(**)
(*Local Alarm*)
VAR
	tyAlmData : tyAlmDat;
	tyInfoData : tyAlmDat;
	tyInfoData1 : tyAlmDat;
	a_tyAlmText : ARRAY[10000..10099] OF tyAlmTxt := [(sAlmText:='New Recipe Not Found In Product Recipe List',sRcyText:='Create New Recipe In Product Setting.'),(sAlmText:='Product Recipe Width Not Match',sRcyText:='Check Product Width And Leader Request Width'),(sAlmText:='New Recipe Not Found In Magazine Recipe List',sRcyText:='Create New Recipe In Magazine Setting.'),(sAlmText:='New Recipe Name Empty',sRcyText:='Request Recipe Name From Leader Is Empty, Check Leader Machine'),6((0)),(sAlmText:='Requested Width Lower Than Minimum Width Limit',sRcyText:='Check The Requested Width Within The Product Limit'),(sAlmText:='Requested Width Larger Than Maxnimum Width Limit',sRcyText:='Check The Requested Width Within The Product Limit'),(sAlmText:='Requested Thickness Larger Than Maximum Thickness Limit',sRcyText:='Check The Requested Thickness Within The Product Limit'),(sAlmText:='Requested Bottom Clearance Larger Than Maximum Bottom Clearance Limit',sRcyText:='Check The Requested Bottom Clearance Within The Product Limit'),(sAlmText:='Requested Top Clearance Larger Than Maximum Top Clearance Limit',sRcyText:='Check The Requested Top Clearance Within The Product Limit'),85((0))];
END_VAR
(**)
(*Local Output*)
VAR
	bUSAllow : BOOL;
	bDSAllow : BOOL;
	tyLeaderInfo : tyLFLeaderInfo;
	bDeleteSendWO : BOOL;
END_VAR
(**)
(*Local Input*)
VAR
	udiRstErr : UDINT := 0;
	bPrep : BOOL := TRUE;
	bEn : BOOL := TRUE;
	bDis : BOOL := FALSE;
	sIPAddr : STRING[15] := '192.168.0.100';
	sMcNm : STRING[30];
	bAWPrep : BOOL := TRUE;
	bAWDis : BOOL;
	bMnlAccData : BOOL;
	bSectionLeader : BOOL;
	sMagRcpNm : STRING[30];
	diWidthLimit : DINT;
	bWidth2Prep : BOOL;
	bUSWidthChkPrep : BOOL;
	bBffrMagRemoved : BOOL;
	bUSWidthChkEn : BOOL;
	bUSWidthChkSen : BOOL;
	bDSWidthChkPrep : BOOL;
	bDSWidthChkEn : BOOL;
	bDSWidthChkSen : BOOL;
	bProdWidthChk : BOOL;
	bUIProdAccData : BOOL;
	bUIProdUpdtData : BOOL;
	bUIMagAccData : BOOL;
	tyCurrProdRcp : tyBoardProperty;
	sCurrMagRcpNm : STRING[30];
	eTimeStat : eTimeAction;
	eTimeStatus : eFBStatus;
	bAccNewRcpCond : BOOL;
	bUpdtNewRcpCond : BOOL;
	bAutoUpdtData : BOOL;
	sInfoMsg : STRING[200];
	bInternalUse : BOOL;
	tyInternalReqProdRcp : tyProdRcpParam;
	bNewBrdEnteredCond : BOOL;
	bOldBrdExitedCond : BOOL;
	bRlsBrd : BOOL;
	tyToLeaderProdRcp : tyProdRcpParam;
	a_bInternalReqProdRcpDiff : ARRAY[0..3] OF BOOL;
	bUpdtProdRcpDiff : BOOL;
	bRlsBrdProdRcpDiff : BOOL;
	sProgNm : STRING[15] := 'AutoRcp';
	bNtSettingsLoadDone : BOOL := TRUE;
	tOnlineChkDlyTm : TIME;
	bManual : BOOL := FALSE;
	bErr : BOOL := FALSE;
	bWarning : BOOL := FALSE;
	bOps : BOOL := FALSE;
	bStandby : BOOL := FALSE;
	eAWStat : eAWAction;
	bFileNotFound : BOOL;
END_VAR
(**)
(*Local*)
VAR
	bRstErr : BOOL;
	udiRstErrOld : UDINT;
	bInitDone : BOOL;
	bInitialDone : BOOL;
	bAutoAccData : BOOL;
	bProdRcpErr : BOOL;
	bMagRcpErr : BOOL;
	bSetTmErr : BOOL;
	bProdAccDataReq : BOOL;
	sReqProdRcpNm : STRING[254];
	diReqProdRcpWidth : DINT;
	bMagAccDataReq : BOOL;
	sReqMagRcpNm : STRING[30];
	usiProdAccDatStep : USINT;
	usiMagAccDatStep : USINT;
	usiProdUpdtDatStep : USINT;
	tyRlsBrdProdRcpNm : tyProdRcpParam;
	bNewBrdEntered : BOOL;
	bOldBrdExited : BOOL;
	i : INT;
	usi : USINT;
	bFollowerInfo : BOOL;
	bDBAOnWOAlign : BOOL;
	tyProRcpCurrRcp : USINT;
	ProdRcpAct : USINT;
	a_bBufferMagPresent : ARRAY[1..4] OF BOOL := [4(FALSE)];
	a_bMagAWWidthDiff : ARRAY[1..4] OF BOOL := [4(FALSE)];
	a_tyBffrStat : ARRAY[1..4] OF tyBffrStat := [4((0))];
	a_sortedMagPriority : ARRAY[1..4] OF USINT;
	a_udiMagAllwMagPresentTm : ARRAY[1..4] OF UDINT;
	ii : INT;
	jj : INT;
	kk : INT;
	usiMag : USINT;
	bCheckNeedMtyMag : BOOL;
	bTravLifWidthDiffBlk : BOOL;
	a_bMagChangOverBlk : ARRAY[1..4] OF BOOL;
	a_bAllwChangeWidth : ARRAY[1..4] OF BOOL;
	a_udiMagAllwGo : ARRAY[1..4] OF UDINT;
	bForceExitMag : BOOL;
	udiMagAllwGo : ARRAY[1..4] OF UDINT;
	a_bCheckDifferent : ARRAY[1..4] OF BOOL;
	udiModuleNum : UDINT := 7201;
	usiPrevChg : USINT;
	usiChg : USINT;
END_VAR
(*local variable*)
VAR
	bTest : BOOL;
	bTest2 : BOOL;
	bMagWriteRetain : BOOL;
	bInitializedFollower1Done : BOOL;
	bOverWriteMagProperties : BOOL;
	bOverWriteTravLifProperties : BOOL;
	bZ1AccNewRcpCondition : BOOL;
	bZ2AccNewRcpCondition : BOOL;
	diRequestedMinSlt : DINT := 3;
	bHermesBAAccpt : BOOL;
	bHermesBFAccpt : BOOL;
	tyHermesBAAccpt : tyHermesBoardAvailable;
	tyHermesBFAccpt : tyHermesBoardForecast;
END_VAR
(*Local Variable for calculation*)
VAR
	rMinslt : REAL;
	rMaxslt : REAL;
	rPitch : REAL;
	rNumInterval : REAL;
	diCalcedPitch : DINT;
	diCalcedMax : DINT;
	diCalcedMin : DINT;
	diModulus : DINT;
	sProdtypeID : STRING[254];
	diProdWidth : DINT;
	diPullerTipHeight : DINT := 45;
END_VAR
(*Rcp Property*)
VAR
	tyCurrReqRcp : tyBoardProperty;
	tyCurrZ1Rcp : tyBoardProperty; (*Mag*)
	a_tyCurrZ2Rcp : ARRAY[1..4] OF tyBoardProperty; (*Mag*)
	a_bRcpLoaded : ARRAY[1..4] OF BOOL;
END_VAR
(*Write Rcp*)
VAR
	a_tyZ2RcpWr : ARRAY[1..4] OF tyBoardProperty; (*Mag1*)
END_VAR
(*from Z2RcpWr to Conveted Mag Properties*)
VAR
	diTravLifPitch : DINT;
	diTravLifWidth : DINT;
	a_tyMagProps : ARRAY[1..4] OF tyMagProperties;
	sWorkOrderId : STRING[80];
END_VAR
(*Save Magazine Rcp*)
VAR
	fbDirCreate1 : fbDirCreate;
	fbDirCreate2 : fbDirCreate;
	fbFileRead1 : fbFileFullRead;
	fbFileRead2 : fbFileFullRead;
	fbFileRead3 : fbFileFullRead;
	fbFileWrite1 : fbFileFullWrite;
	fbFileWrite2 : fbFileFullWrite;
	fbFileWrite3 : fbFileFullWrite;
END_VAR
(*WeFab*)
VAR
	a_tyAutoRcpFollower1 : tyProdRcpParam := (diWidthInUM:=100000);
	a_tyAutoRcpInternal : ARRAY[1..3] OF tyProdRcpParam;
	tyCurrReqMagRcp : tyProdRcpParam;
	a_tyAutoRcpInternalWr : ARRAY[1..3] OF tyProdRcpParam;
	tyCurrZ1Rcp1_Int : tyProdRcpParam;
END_VAR
```

Listed in the project but not available here: Logical/UI/UI/Act_LinkAction.st, Logical/UI/UI/Cyclic.st, Logical/UI/UI/Act_Action.st, Logical/UI/UI/Act_Main/Act_Main_C0007.st, Logical/UI/UI/Act_Main/Act_Main_P0002.st, Logical/UI/UI/Act_Main/Act_Main_P0300.st, Logical/UI/UI/Act_Main/Act_Main_P0934.st, Logical/UI/UI/Act_Main/Act_Main_P0937.st, Logical/UI/UI/Act_Main/Act_Main_P1000.st, Logical/UI/UI/Act_Main/Act_Main_P1080.st, Logical/UI/UI/Act_Background.st, Logical/UI/UI/Act_Background/Action/C0001, Logical/UI/UI/Act_Background/Action/C0002, Logical/UI/UI/Act_Background/Action/C0003, Logical/UI/UI/Act_Background/Action/C0004, Logical/UI/UI/Act_Background/Action/C0006, Logical/UI/UI/Act_Background/Action/C0008, Logical/UI/UI/Act_Background/Action/C0009, Logical/UI/UI/Act_Background/Action/C0010, Logical/UI/UI/Act_Background/Action/P0100, Logical/UI/UI/Act_Background/Action/P0200/Act_OptP0200RcyMsg.st, Logical/UI/UI/Act_Background/Action/P0202/Act_OptP0202Navi.st, Logical/UI/UI/Act_Background/Action/P0202/Act_OptP0202ChgPage.st, Logical/UI/UI/Act_Background/Action/P0202/Act_OptP0202RstMnl.st, Logical/UI/UI/Act_Background/Action/P0203/Act_OptP0203Navi.st, Logical/UI/UI/Act_Background/Action/P0203/Act_OptP0203ChgPage.st, Logical/UI/UI/Act_Background/Action/P0203/Act_OptP0203RstMnl.st, Logical/UI/UI/Act_Background/Action/P0800/Act_OptP0800Table1.st, Logical/UI/UI/Act_Background/Action/P0800/Act_OptP0800Table2.st, Logical/UI/UI/Act_Background/Action/P0800/Act_OptP0800Table3.st, Logical/UI/UI/Act_Background/Action/P0921/Act_OptP0921InletShutterFBStat.st, Logical/UI/UI/Act_Background/Action/P0921/Act_OptP0921OutletShutterFBStat.st, Logical/UI/UI/Act_Background/Action/P0921/Act_OptP0921OutletShutterDC.st, Logical/UI/UI/Act_Background/Action/P0950/Act_OptP0950SimuMod.st, Logical/UI/UI/Act_Background/Action/P1021/Act_OptP1021IPAddr.st, Logical/UI/UI/Act_Background/Action/P1021/Act_OptP1021SubnetMask.st, Logical/UI/UI/Act_Background/Action/P1021/Act_OptP1021DHCPSetting.st, Logical/UI/UI/Act_Background/Action/P1026/Act_OptP1026Navi.st, Logical/UI/UI/Act_Background/Action/P1026/Act_OptP1026FullMask.st, Logical/UI/UI/Act_Background/Action/P1026/Act_OptP1026Mnl.st, Logical/UI/UI/Act_Background/Action/P1026/Act_OptP1026TravFBStat.st, Logical/UI/UI/Act_Background/Action/P1026/Act_OptP1026TravMask.st, Logical/UI/UI/Act_Background/Action/P1026/Act_OptP1026TravKeypad.st, Logical/UI/UI/Act_Background/Action/P1026/Act_OptP1026TravRstMnl.st, Logical/UI/UI/Act_Background/Action/P1026/Act_OptP1026LifterFBStat.st, Logical/UI/UI/Act_Background/Action/P1026/Act_OptP1026LifterMask.st, Logical/UI/UI/Act_Background/Action/P1026/Act_OptP1026LifterKeypad.st, Logical/UI/UI/Act_Background/Action/P1031/Act_OptP1031Navi.st, Logical/UI/UI/Act_Background/Action/P1031/Act_OptP1031Mnl.st, Logical/UI/UI/Act_Background/Action/P1031/Act_OptP1031TravFBStat.st, Logical/UI/UI/Act_Background/Action/P1031/Act_OptP1031TravKeypad.st, Logical/UI/UI/Act_Background/Action/P1031/Act_OptP1031LifterFBStat.st, Logical/Startup/Startup/Act_Main/Act_Main_UsrFolder.st, Logical/Startup/Startup/Act_Main/Act_Main_GetHWInfo.st, Logical/Startup/Startup/Act_Main/Act_Main_LibVer.st, Logical/Startup/Startup/Act_Main/Act_Main_Parameter.st, Logical/Startup/Startup/Act_Main/Act_Main_UsrMgmt.st, Logical/Startup/Startup/Act_Main/Act_Main_SetupUI.st, Logical/Startup/Startup/Act_Main/Act_Main_Done.st, Logical/General, Logical/RstErr, Logical/Buffer/Buffer.typ, Logical/Buffer/Buffer1.var, Logical/Buffer/Buffer2.var, Logical/Buffer/Buffer3.var, Logical/SMEMA/SMEMA.typ, Logical/SMEMA/USSMEMA1.var, Logical/SMEMA/USSMEMA2.var, Logical/SMEMA/USSMEMA3.var, Logical/Pneu/Pneu.typ, Logical/Pneu/Pneu2SenOutShutter.var, Logical/Pneu/SelClamp/Pneu2SenSelClamp1.var, Logical/Pneu/SelClamp/Pneu2SenSelClamp2.var, Logical/Pneu/SelClamp/Pneu2SenSelClamp3.var, Logical/Pneu/MagSafetyBar/Pneu2SenMag1SafetyBar.var, Logical/Pneu/MagSafetyBar/Pneu2SenMag2SafetyBar.var, Logical/Pneu/MagSafetyBar/Pneu2SenMag3SafetyBar.var, Logical/Pneu/Trolley/PneuExtSenTrolley/Act_LinkEn.st, Logical/Pneu/Trolley/PneuExtSenTrolley/Act_Link.st, Logical/Pneu/Trolley/PneuExtSenTrolley/Cyclic.st, Logical/Pneu/Trolley/PneuExtSenTrolley/Act_RstErr.st, Logical/Pneu/Trolley/PneuExtSenTrolley/Act_Initial.st, Logical/Pneu/Trolley/PneuExtSenTrolley/Act_Action.st, Logical/Pneu/Trolley/PneuExtSenTrolley/Act_Main.st, Logical/Pneu/Pneu2SenInShutter3.var, Logical/Conv/PullConv/Act_LinkEn.st, Logical/Conv/PullConv/Cyclic.st, Logical/Conv/PullConv/Act_RstErr.st, Logical/Conv/PullConv/Act_InitLocal.st, Logical/Conv/PullConv/Act_Initial.st, Logical/Conv/PullConv/Act_Action.st, Logical/Conv/PullConv/Act_Background.st, Logical/MagConv/MagConv2Clp1.var, Logical/MagConv/MagConv2Clp2.var, Logical/MagConv/MagConv2Clp3.var, Logical/MagConv/MagConv2Clp3/Init.st, Logical/MagConv/MagConv2Clp3/InputRef_Link.var, Logical/MagConv/MagConv2Clp3/Act_LinkEn.st, Logical/MagConv/MagConv2Clp3/Cyclic.st, Logical/MagConv/MagConv2Clp3/Act_RstErr.st, Logical/MagConv/MagConv2Clp3/Act_InitLocal.st, Logical/MagConv/MagConv2Clp3/Act_Initial.st, Logical/MagConv/MagConv2Clp3/Act_Main.st, Logical/MagConv/MagConv2Clp3/Act_Action.st, Logical/MagConv/MagConv2Clp3/Act_Alarm.st, Logical/MagConv/MagConv2Clp3/InputRef.var, Logical/CANOpenServo/CANOpenServo.typ, Logical/CANOpenServo/Lifter/Lifter.typ, Logical/CANOpenServo/Lifter/LifterBtm.var, Logical/CANOpenServo/PullerPusher/PullerPusher.typ, Logical/DOutput/DOutput/Init.st, Logical/DOutput/DOutput/Act_LinkAction.st, Logical/DOutput/DOutput/Cyclic.st, Logical/DOutput/DOutput/Act_Initial.st, Logical/DOutput/DOutput/Act_Action.st, Logical/DOutput/DOutput/Act_Main.st, Logical/Hermes/Hermes.typ, Logical/Hermes/DSHermesB/Act_LinkEn.st, Logical/Hermes/DSHermesB/Cyclic.st, Logical/Hermes/DSHermesB/Act_RstErr.st, Logical/Hermes/DSHermesB/Act_InitLocal.st, Logical/Hermes/DSHermesB/Act_Initial.st, Logical/Hermes/DSHermesB/Act_Action.st, Logical/Hermes/DSHermesB/Act_Main.st, Logical/Hermes/DSHermesB/Act_Background.st, Logical/Hermes/DSHermesB/Act_Background_TCPCreateSvr.st, Logical/Hermes/DSHermesB/Act_Background_TCPListen.st, Logical/Hermes/DSHermesB/Act_Background_TCPRcv.st, Logical/Hermes/DSHermesB/Act_Background_NotificationRcv.st, Logical/Hermes/DSHermesB/Act_Background_IllegalMsg.st, Logical/Hermes/DSHermesB/Act_Background_ChkParamRcv.st, Logical/Hermes/DSHermesB/Act_Background_SequenceTO.st, Logical/Hermes/DSHermesB/Act_Background_ChkAlive.st, Logical/Hermes/DSHermesB/Act_Background_ChkAliveSendPing.st, Logical/Hermes/DSHermesB/Act_Background_ChkAliveRcvPing.st, Logical/Hermes/DSHermesB/Act_Background_ChgConfig.st, Logical/Hermes/DSHermesB/Act_Background_NotificationSnd.st, Logical/Hermes/DSHermesB/Act_Background_TCPSend.st, Logical/Hermes/DSHermesB/Act_Background_TCPCloseSvr.st, Logical/Hermes/DSHermesB/Act_Background_TCPCloseClnt.st, Logical/Hermes/DSHermesB/Act_Background_Stop.st, Logical/Hermes/DSHermesB/Act_Background_Log.st, Logical/Hermes/DSHermesB/Act_Background_Err.st, Logical/Hermes/DSHermesB/Act_Main_Disable.st, Logical/Hermes/DSHermesB/Act_CombineErr.st, Logical/Hermes/RmtHermes/Init.st, Logical/Hermes/RmtHermes/Act_InitGlobal.st, Logical/Hermes/RmtHermes/InputRef_Link.var, Logical/Hermes/RmtHermes/Act_LinkAction.st, Logical/Hermes/RmtHermes/Act_LinkEn.st, Logical/Hermes/RmtHermes/Act_Link.st, Logical/Hermes/RmtHermes/Cyclic.st, Logical/Hermes/RmtHermes/Act_RstErr.st, Logical/Hermes/RmtHermes/Act_InitLocal.st, Logical/Hermes/RmtHermes/Act_Initial.st, Logical/Hermes/RmtHermes/Act_Action.st, Logical/Hermes/RmtHermes/Act_Main.st, Logical/Hermes/RmtHermes/Act_Background.st, Logical/Hermes/RmtHermes/Act_Background_ProcessData.st, Logical/Hermes/RmtHermes/Act_Background_TCPCreateSvr.st, Logical/Hermes/RmtHermes/Act_Background_TCPListen.st, Logical/Hermes/RmtHermes/Act_Background_TCPRcv.st, Logical/Hermes/RmtHermes/Act_Background_NotificationRcv.st, Logical/Hermes/RmtHermes/Act_Background_IllegalMsg.st, Logical/Hermes/RmtHermes/Act_Background_UpdtConfig.st, Logical/Hermes/RmtHermes/Act_Background_SendConfig.st, Logical/Hermes/RmtHermes/Act_Background_NotificationSnd.st, Logical/Hermes/RmtHermes/Act_Background_TCPSend.st, Logical/Hermes/RmtHermes/Act_Background_TCPCloseSvr.st, Logical/Hermes/RmtHermes/Act_Background_TCPCloseClnt.st, Logical/Hermes/RmtHermes/Act_Background_Stop.st, Logical/Hermes/RmtHermes/Act_Background_Log.st, Logical/Hermes/RmtHermes/Act_Background_Err.st, Logical/Hermes/RmtHermes/Act_Main_Disable.st, Logical/Hermes/RmtHermes/Act_CombineErr.st, Logical/Hermes/RmtHermes/InputRef.var, Logical/Hermes/RmtHermes/Local.var, Logical/Operations/Operations.typ, Logical/Operations/Ops.var, Logical/Operations/OpsMagConvLD1/Sequence/Act_OpsInitial.st, Logical/Operations/OpsMagConvLD1/Sequence/Act_OpsRst.st, Logical/Operations/OpsMagConvLD1/Sequence/Act_LogStep.st, Logical/AGVCom/AGV.var, Logical/AGVCom/AGV/Act_LinkAction.st, Logical/AGVCom/AGV/Act_LinkEn.st, Logical/AGVCom/AGV/Cyclic.st, Logical/AGVCom/AGV/Act_RstErr.st, Logical/AGVCom/AGV/Act_Action.st, Logical/AGVCom/AGV1.var, Logical/AGVCom/AGV2.var, Logical/AGVCom/AGV3.var, Logical/Simulation/Simulation.typ, Logical/Simulation/Simu.var, Logical/Simulation/Simu, Logical/SOT/SOT.typ, Logical/SOT/USSOT1.var, Logical/SOT/DSSOT1.var, Logical/SOT/USSOT2.var, Logical/SOT/DSSOT2.var, Logical/SOT/DSSOT3.var, Logical/Machine/Machine.var, Logical/Machine/Machine1/Act_RstErr.st, Logical/Machine/Machine1/Act_InitLocal.st, Logical/Machine/Machine1/Act_Initial.st, Logical/Machine/Machine1/Act_Background.st, Logical/Machine/Machine1/Act_AlarmInfo1.st, Logical/USBBarcodeRdr/BarcodeRdr/Act_CombineErr.st, Logical/RS232/DVFrame/Frame/Act_LinkEn.st, Logical/RS232/DVFrame/Frame/Act_RstErr.st, Logical/RS232/DVFrame/Frame/Act_CombineErr.st, Logical/AutoRcp/AutoRcp.typ, Logical/AutoRcp/AutoRcp/Act_LinkAction.st, Logical/AutoRcp/AutoRcp/Act_RstErr.st, Logical/AutoRcp/AutoRcp/Act_Action.st, Logical/AutoRcp/AutoRcp/Act_Main_Disable.st, Logical/AutoRcp/AutoRcp/Act_Alarm.st
